LIN {X 0,Y 439.372,Z 569.757,A -85,B 0,C 180,E1 -9212.03,E2 -9212.03} C_VEL
LIN {X 0,Y 439.398,Z 569.751,A -85,B 0,C 180,E1 -9215.34,E2 -9215.34} C_VEL
LIN {X 0,Y 439.39,Z 569.756,A -85,B 0,C 180,E1 -9218.594,E2 -9218.594} C_VEL
LIN {X 0,Y 439.391,Z 569.751,A -85,B 0,C 180,E1 -9221.256,E2 -9221.256} C_VEL
LIN {X 0,Y 439.407,Z 569.752,A -85,B 0,C 180,E1 -9224.728,E2 -9224.728} C_VEL
LIN {X 0,Y 439.399,Z 569.751,A -85,B 0,C 180,E1 -9227.795,E2 -9227.795} C_VEL
LIN {X 0,Y 439.438,Z 569.749,A -85,B 0,C 180,E1 -9230.228,E2 -9230.228} C_VEL
LIN {X 0,Y 439.374,Z 569.754,A -85,B 0,C 180,E1 -9233.712,E2 -9233.712} C_VEL
LIN {X 0,Y 439.373,Z 569.756,A -85,B 0,C 180,E1 -9237.053,E2 -9237.053} C_VEL
LIN {X 0,Y 439.383,Z 569.755,A -85,B 0,C 180,E1 -9240.274,E2 -9240.274} C_VEL
LIN {X 0,Y 439.429,Z 569.747,A -85,B 0,C 180,E1 -9243.396,E2 -9243.396} C_VEL
LIN {X 0,Y 439.387,Z 569.755,A -85,B 0,C 180,E1 -9246.429,E2 -9246.429} C_VEL
LIN {X 0,Y 439.388,Z 569.751,A -85,B 0,C 180,E1 -9249.396,E2 -9249.396} C_VEL
LIN {X 0,Y 439.431,Z 569.749,A -85,B 0,C 180,E1 -9252.309,E2 -9252.309} C_VEL
LIN {X 0,Y 439.447,Z 569.746,A -85,B 0,C 180,E1 -9255.173,E2 -9255.173} C_VEL
LIN {X 0,Y 439.507,Z 569.738,A -85,B 0,C 180,E1 -9258.001,E2 -9258.001} C_VEL
LIN {X 0,Y 439.547,Z 569.733,A -85,B 0,C 180,E1 -9261.725,E2 -9261.725} C_VEL
LIN {X 0,Y 439.621,Z 569.726,A -85,B 0,C 180,E1 -9264.495,E2 -9264.495} C_VEL
LIN {X 0,Y 439.635,Z 569.724,A -85,B 0,C 180,E1 -9268.167,E2 -9268.167} C_VEL
LIN {X 0,Y 439.63,Z 569.725,A -85,B 0,C 180,E1 -9268.568,E2 -9268.568} C_VEL
LIN {X 0,Y 442.794,Z 580.936,A -85,B 0,C 180,E1 -9269.301,E2 -9269.301} C_VEL
LIN {X 0,Y 442.766,Z 587.106,A -85,B 0,C 180,E1 -9269.714,E2 -9269.714} C_VEL
LIN {X 0,Y 442.691,Z 589.675,A -85,B 0,C 180,E1 -9269.904,E2 -9269.904} C_VEL
LIN {X 0,Y 441.903,Z 594.784,A -85,B 0,C 180,E1 -9270.276,E2 -9270.276} C_VEL
LIN {X 0,Y 438.786,Z 602.936,A -85,B 0,C 180,E1 -9270.891,E2 -9270.891} C_VEL
LIN {X 0,Y 435.571,Z 610.599,A -85,B 0,C 180,E1 -9271.598,E2 -9271.598} C_VEL
LIN {X 0,Y 434.642,Z 614.939,A -85,B 0,C 180,E1 -9272.11,E2 -9272.11} C_VEL
LIN {X 0,Y 433.977,Z 624.554,A -85,B 0,C 180,E1 -9273.481,E2 -9273.481} C_VEL
LIN {X 0,Y 433.566,Z 632.408,A -85,B 0,C 180,E1 -9274.881,E2 -9274.881} C_VEL
LIN {X 0,Y 433.204,Z 637.758,A -85,B 0,C 180,E1 -9276.052,E2 -9276.052} C_VEL
LIN {X 0,Y 432.906,Z 642.988,A -85,B 0,C 180,E1 -9277.461,E2 -9277.461} C_VEL
LIN {X 0,Y 432.602,Z 647.086,A -85,B 0,C 180,E1 -9278.877,E2 -9278.877} C_VEL
LIN {X 0,Y 432.379,Z 650.136,A -85,B 0,C 180,E1 -9280.299,E2 -9280.299} C_VEL
LIN {X 0,Y 432.284,Z 651.639,A -85,B 0,C 180,E1 -9281.249,E2 -9281.249} C_VEL
LIN {X 0,Y 432.251,Z 653.107,A -85,B 0,C 180,E1 -9282.7,E2 -9282.7} C_VEL
LIN {X 0,Y 432.204,Z 653.639,A -85,B 0,C 180,E1 -9284.117,E2 -9284.117} C_VEL
LIN {X 0,Y 432.223,Z 653.484,A -85,B 0,C 180,E1 -9285.079,E2 -9285.079} C_VEL
LIN {X 0,Y 432.331,Z 652.582,A -85,B 0,C 180,E1 -9286.443,E2 -9286.443} C_VEL
LIN {X 0,Y 432.509,Z 650.537,A -85,B 0,C 180,E1 -9287.982,E2 -9287.982} C_VEL
LIN {X 0,Y 432.853,Z 646.995,A -85,B 0,C 180,E1 -9289.66,E2 -9289.66} C_VEL
LIN {X 0,Y 433.263,Z 641.799,A -85,B 0,C 180,E1 -9291.405,E2 -9291.405} C_VEL
LIN {X 0,Y 433.769,Z 635.934,A -85,B 0,C 180,E1 -9292.882,E2 -9292.882} C_VEL
LIN {X 0,Y 434.305,Z 628.458,A -85,B 0,C 180,E1 -9294.37,E2 -9294.37} C_VEL
LIN {X 0,Y 434.941,Z 620.541,A -85,B 0,C 180,E1 -9295.636,E2 -9295.636} C_VEL
LIN {X 0,Y 435.577,Z 611.178,A -85,B 0,C 180,E1 -9296.857,E2 -9296.857} C_VEL
LIN {X 0,Y 436.16,Z 600.306,A -85,B 0,C 180,E1 -9297.988,E2 -9297.988} C_VEL
LIN {X 0,Y 436.788,Z 589.714,A -85,B 0,C 180,E1 -9298.861,E2 -9298.861} C_VEL
LIN {X 0,Y 436.842,Z 584.716,A -85,B 0,C 180,E1 -9299.218,E2 -9299.218} C_VEL
LIN {X 0,Y 433.122,Z 573.093,A -85,B 0,C 180,E1 -9300.097,E2 -9300.097} C_VEL
LIN {X 0,Y 432.389,Z 570.629,A -85,B 0,C 180,E1 -9300.255,E2 -9300.255} C_VEL
LIN {X 0,Y 432.353,Z 570.628,A -85,B 0,C 180,E1 -9304.003,E2 -9304.003} C_VEL
LIN {X 0,Y 432.328,Z 570.635,A -85,B 0,C 180,E1 -9307.198,E2 -9307.198} C_VEL
LIN {X 0,Y 432.436,Z 570.815,A -85,B 0,C 180,E1 -9308.895,E2 -9308.895} C_VEL
LIN {X 0,Y 433.241,Z 576.214,A -85,B 0,C 180,E1 -9311.069,E2 -9311.069} C_VEL
LIN {X 0,Y 433.258,Z 582.668,A -85,B 0,C 180,E1 -9313.627,E2 -9313.627} C_VEL
LIN {X 0,Y 433.14,Z 590.995,A -85,B 0,C 180,E1 -9316.898,E2 -9316.898} C_VEL
LIN {X 0,Y 432.831,Z 599.434,A -85,B 0,C 180,E1 -9320.219,E2 -9320.219} C_VEL
LIN {X 0,Y 432.697,Z 606.671,A -85,B 0,C 180,E1 -9323.061,E2 -9323.061} C_VEL
LIN {X 0,Y 432.492,Z 615.337,A -85,B 0,C 180,E1 -9326.462,E2 -9326.462} C_VEL
LIN {X 0,Y 432.248,Z 623.677,A -85,B 0,C 180,E1 -9329.733,E2 -9329.733} C_VEL
LIN {X 0,Y 432.206,Z 625.589,A -85,B 0,C 180,E1 -9330.479,E2 -9330.479} C_VEL
LIN {X 0,Y 435.447,Z 641.385,A -85,B 0,C 180,E1 -9331.111,E2 -9331.111} C_VEL
LIN {X 0,Y 435.762,Z 646.126,A -85,B 0,C 180,E1 -9331.329,E2 -9331.329} C_VEL
LIN {X 0,Y 435.232,Z 658.171,A -85,B 0,C 180,E1 -9331.96,E2 -9331.96} C_VEL
LIN {X 0,Y 434.708,Z 669.886,A -85,B 0,C 180,E1 -9332.769,E2 -9332.769} C_VEL
LIN {X 0,Y 434.076,Z 680.526,A -85,B 0,C 180,E1 -9333.691,E2 -9333.691} C_VEL
LIN {X 0,Y 433.476,Z 690.924,A -85,B 0,C 180,E1 -9334.812,E2 -9334.812} C_VEL
LIN {X 0,Y 432.897,Z 700.253,A -85,B 0,C 180,E1 -9336.055,E2 -9336.055} C_VEL
LIN {X 0,Y 432.385,Z 708.024,A -85,B 0,C 180,E1 -9337.318,E2 -9337.318} C_VEL
LIN {X 0,Y 432.035,Z 715.276,A -85,B 0,C 180,E1 -9338.781,E2 -9338.781} C_VEL
LIN {X 0,Y 431.673,Z 721.759,A -85,B 0,C 180,E1 -9340.461,E2 -9340.461} C_VEL
LIN {X 0,Y 431.436,Z 726.172,A -85,B 0,C 180,E1 -9341.971,E2 -9341.971} C_VEL
LIN {X 0,Y 431.358,Z 728.335,A -85,B 0,C 180,E1 -9342.947,E2 -9342.947} C_VEL
LIN {X 0,Y 431.26,Z 730.235,A -85,B 0,C 180,E1 -9344.043,E2 -9344.043} C_VEL
LIN {X 0,Y 431.221,Z 731.301,A -85,B 0,C 180,E1 -9344.885,E2 -9344.885} C_VEL
LIN {X 0,Y 431.171,Z 732.08,A -85,B 0,C 180,E1 -9345.848,E2 -9345.848} C_VEL
LIN {X 0,Y 431.179,Z 732.449,A -85,B 0,C 180,E1 -9346.81,E2 -9346.81} C_VEL
LIN {X 0,Y 431.29,Z 732.372,A -85,B 0,C 180,E1 -9347.876,E2 -9347.876} C_VEL
LIN {X 0,Y 431.271,Z 731.013,A -85,B 0,C 180,E1 -9349.674,E2 -9349.674} C_VEL
LIN {X 0,Y 431.343,Z 729.708,A -85,B 0,C 180,E1 -9350.623,E2 -9350.623} C_VEL
LIN {X 0,Y 431.546,Z 726.899,A -85,B 0,C 180,E1 -9352.044,E2 -9352.044} C_VEL
LIN {X 0,Y 431.711,Z 723.065,A -85,B 0,C 180,E1 -9353.457,E2 -9353.457} C_VEL
LIN {X 0,Y 431.952,Z 718.085,A -85,B 0,C 180,E1 -9354.866,E2 -9354.866} C_VEL
LIN {X 0,Y 432.307,Z 711.79,A -85,B 0,C 180,E1 -9356.272,E2 -9356.272} C_VEL
LIN {X 0,Y 432.829,Z 703.98,A -85,B 0,C 180,E1 -9357.674,E2 -9357.674} C_VEL
LIN {X 0,Y 433.386,Z 696.051,A -85,B 0,C 180,E1 -9358.839,E2 -9358.839} C_VEL
LIN {X 0,Y 434.041,Z 686.397,A -85,B 0,C 180,E1 -9360,E2 -9360} C_VEL
LIN {X 0,Y 434.7,Z 675.647,A -85,B 0,C 180,E1 -9361.043,E2 -9361.043} C_VEL
LIN {X 0,Y 435.374,Z 663.66,A -85,B 0,C 180,E1 -9361.966,E2 -9361.966} C_VEL
LIN {X 0,Y 436.015,Z 650.788,A -85,B 0,C 180,E1 -9362.714,E2 -9362.714} C_VEL
LIN {X 0,Y 436.08,Z 643.477,A -85,B 0,C 180,E1 -9363.061,E2 -9363.061} C_VEL
LIN {X 0,Y 433.461,Z 631.54,A -85,B 0,C 180,E1 -9363.603,E2 -9363.603} C_VEL
LIN {X 0,Y 432.321,Z 627.329,A -85,B 0,C 180,E1 -9363.787,E2 -9363.787} C_VEL
LIN {X 0,Y 432.607,Z 622.657,A -85,B 0,C 180,E1 -9365.594,E2 -9365.594} C_VEL
LIN {X 0,Y 432.829,Z 614.137,A -85,B 0,C 180,E1 -9368.874,E2 -9368.874} C_VEL
LIN {X 0,Y 433.025,Z 606.775,A -85,B 0,C 180,E1 -9371.705,E2 -9371.705} C_VEL
LIN {X 0,Y 433.189,Z 599.173,A -85,B 0,C 180,E1 -9374.565,E2 -9374.565} C_VEL
LIN {X 0,Y 433.297,Z 591.196,A -85,B 0,C 180,E1 -9377.462,E2 -9377.462} C_VEL
LIN {X 0,Y 433.431,Z 582.92,A -85,B 0,C 180,E1 -9380.403,E2 -9380.403} C_VEL
LIN {X 0,Y 433.298,Z 575.774,A -85,B 0,C 180,E1 -9382.91,E2 -9382.91} C_VEL
LIN {X 0,Y 432.358,Z 570.636,A -85,B 0,C 180,E1 -9384.762,E2 -9384.762} C_VEL
LIN {X 0,Y 432.387,Z 570.629,A -85,B 0,C 180,E1 -9387.072,E2 -9387.072} C_VEL
LIN {X 0,Y 432.362,Z 570.631,A -85,B 0,C 180,E1 -9390.516,E2 -9390.516} C_VEL
LIN {X 0,Y 432.354,Z 570.631,A -85,B 0,C 180,E1 -9394.005,E2 -9394.005} C_VEL
LIN {X 0,Y 432.329,Z 570.633,A -85,B 0,C 180,E1 -9397.2,E2 -9397.2} C_VEL
LIN {X 0,Y 432.353,Z 570.629,A -85,B 0,C 180,E1 -9400.184,E2 -9400.184} C_VEL
LIN {X 0,Y 432.361,Z 570.63,A -85,B 0,C 180,E1 -9403.056,E2 -9403.056} C_VEL
LIN {X 0,Y 432.374,Z 570.63,A -85,B 0,C 180,E1 -9405.66,E2 -9405.66} C_VEL
LIN {X 0,Y 432.377,Z 570.803,A -85,B 0,C 180,E1 -9407.351,E2 -9407.351} C_VEL
LIN {X 0,Y 434.187,Z 579.301,A -85,B 0,C 180,E1 -9410.257,E2 -9410.257} C_VEL
LIN {X 0,Y 435.681,Z 587.385,A -85,B 0,C 180,E1 -9412.837,E2 -9412.837} C_VEL
LIN {X 0,Y 435.534,Z 593.083,A -85,B 0,C 180,E1 -9414.486,E2 -9414.486} C_VEL
LIN {X 0,Y 434.642,Z 604.82,A -85,B 0,C 180,E1 -9417.752,E2 -9417.752} C_VEL
LIN {X 0,Y 433.929,Z 616.968,A -85,B 0,C 180,E1 -9420.998,E2 -9420.998} C_VEL
LIN {X 0,Y 433.289,Z 629.663,A -85,B 0,C 180,E1 -9424.287,E2 -9424.287} C_VEL
LIN {X 0,Y 432.691,Z 643.56,A -85,B 0,C 180,E1 -9427.794,E2 -9427.794} C_VEL
LIN {X 0,Y 432.277,Z 657.625,A -85,B 0,C 180,E1 -9431.272,E2 -9431.272} C_VEL
LIN {X 0,Y 432.086,Z 665.28,A -85,B 0,C 180,E1 -9433.15,E2 -9433.15} C_VEL
LIN {X 0,Y 433.733,Z 681.12,A -85,B 0,C 180,E1 -9433.658,E2 -9433.658} C_VEL
LIN {X 0,Y 434.619,Z 693.584,A -85,B 0,C 180,E1 -9434.226,E2 -9434.226} C_VEL
LIN {X 0,Y 435.052,Z 699.186,A -85,B 0,C 180,E1 -9434.542,E2 -9434.542} C_VEL
LIN {X 0,Y 434.161,Z 715.758,A -85,B 0,C 180,E1 -9435.59,E2 -9435.59} C_VEL
LIN {X 0,Y 433.491,Z 727,A -85,B 0,C 180,E1 -9436.507,E2 -9436.507} C_VEL
LIN {X 0,Y 432.961,Z 737.61,A -85,B 0,C 180,E1 -9437.581,E2 -9437.581} C_VEL
LIN {X 0,Y 432.469,Z 747.017,A -85,B 0,C 180,E1 -9438.756,E2 -9438.756} C_VEL
LIN {X 0,Y 431.986,Z 756.151,A -85,B 0,C 180,E1 -9440.165,E2 -9440.165} C_VEL
LIN {X 0,Y 431.714,Z 763.519,A -85,B 0,C 180,E1 -9441.576,E2 -9441.576} C_VEL
LIN {X 0,Y 431.516,Z 769.377,A -85,B 0,C 180,E1 -9442.985,E2 -9442.985} C_VEL
LIN {X 0,Y 431.451,Z 773.978,A -85,B 0,C 180,E1 -9444.392,E2 -9444.392} C_VEL
LIN {X 0,Y 431.397,Z 776.404,A -85,B 0,C 180,E1 -9445.329,E2 -9445.329} C_VEL
LIN {X 0,Y 431.377,Z 778.39,A -85,B 0,C 180,E1 -9446.264,E2 -9446.264} C_VEL
LIN {X 0,Y 431.407,Z 779.895,A -85,B 0,C 180,E1 -9447.2,E2 -9447.2} C_VEL
LIN {X 0,Y 431.405,Z 780.964,A -85,B 0,C 180,E1 -9448.134,E2 -9448.134} C_VEL
LIN {X 0,Y 431.402,Z 781.628,A -85,B 0,C 180,E1 -9449.067,E2 -9449.067} C_VEL
LIN {X 0,Y 431.382,Z 781.873,A -85,B 0,C 180,E1 -9450.001,E2 -9450.001} C_VEL
LIN {X 0,Y 431.401,Z 781.664,A -85,B 0,C 180,E1 -9450.934,E2 -9450.934} C_VEL
LIN {X 0,Y 431.407,Z 781.049,A -85,B 0,C 180,E1 -9451.868,E2 -9451.868} C_VEL
LIN {X 0,Y 431.406,Z 780.029,A -85,B 0,C 180,E1 -9452.802,E2 -9452.802} C_VEL
LIN {X 0,Y 431.36,Z 778.542,A -85,B 0,C 180,E1 -9453.737,E2 -9453.737} C_VEL
LIN {X 0,Y 431.445,Z 775.484,A -85,B 0,C 180,E1 -9455.141,E2 -9455.141} C_VEL
LIN {X 0,Y 431.445,Z 771.315,A -85,B 0,C 180,E1 -9456.548,E2 -9456.548} C_VEL
LIN {X 0,Y 431.65,Z 764.913,A -85,B 0,C 180,E1 -9458.191,E2 -9458.191} C_VEL
LIN {X 0,Y 431.93,Z 757.897,A -85,B 0,C 180,E1 -9459.601,E2 -9459.601} C_VEL
LIN {X 0,Y 432.355,Z 749.061,A -85,B 0,C 180,E1 -9461.012,E2 -9461.012} C_VEL
LIN {X 0,Y 432.872,Z 739.007,A -85,B 0,C 180,E1 -9462.305,E2 -9462.305} C_VEL
LIN {X 0,Y 433.409,Z 728.753,A -85,B 0,C 180,E1 -9463.359,E2 -9463.359} C_VEL
LIN {X 0,Y 434.093,Z 717.383,A -85,B 0,C 180,E1 -9464.295,E2 -9464.295} C_VEL
LIN {X 0,Y 434.676,Z 705.557,A -85,B 0,C 180,E1 -9465.053,E2 -9465.053} C_VEL
LIN {X 0,Y 434.802,Z 696.334,A -85,B 0,C 180,E1 -9465.529,E2 -9465.529} C_VEL
LIN {X 0,Y 433.813,Z 685.114,A -85,B 0,C 180,E1 -9466.063,E2 -9466.063} C_VEL
LIN {X 0,Y 432.601,Z 671.595,A -85,B 0,C 180,E1 -9466.526,E2 -9466.526} C_VEL
LIN {X 0,Y 432.071,Z 666.093,A -85,B 0,C 180,E1 -9466.682,E2 -9466.682} C_VEL
LIN {X 0,Y 432.394,Z 652.62,A -85,B 0,C 180,E1 -9469.958,E2 -9469.958} C_VEL
LIN {X 0,Y 432.844,Z 638.506,A -85,B 0,C 180,E1 -9473.442,E2 -9473.442} C_VEL
LIN {X 0,Y 433.472,Z 624.3,A -85,B 0,C 180,E1 -9476.999,E2 -9476.999} C_VEL
LIN {X 0,Y 434.144,Z 610.513,A -85,B 0,C 180,E1 -9480.521,E2 -9480.521} C_VEL
LIN {X 0,Y 434.876,Z 596.628,A -85,B 0,C 180,E1 -9484.167,E2 -9484.167} C_VEL
LIN {X 0,Y 435.346,Z 587.383,A -85,B 0,C 180,E1 -9486.678,E2 -9486.678} C_VEL
LIN {X 0,Y 434.429,Z 581.267,A -85,B 0,C 180,E1 -9488.446,E2 -9488.446} C_VEL
LIN {X 0,Y 432.378,Z 570.63,A -85,B 0,C 180,E1 -9491.727,E2 -9491.727} C_VEL
LIN {X 0,Y 432.339,Z 570.634,A -85,B 0,C 180,E1 -9494.347,E2 -9494.347} C_VEL
LIN {X 0,Y 432.325,Z 570.635,A -85,B 0,C 180,E1 -9497.016,E2 -9497.016} C_VEL
LIN {X 0,Y 432.346,Z 570.631,A -85,B 0,C 180,E1 -9499.82,E2 -9499.82} C_VEL
LIN {X 0,Y 432.32,Z 570.632,A -85,B 0,C 180,E1 -9503.023,E2 -9503.023} C_VEL
LIN {X 0,Y 432.365,Z 570.629,A -85,B 0,C 180,E1 -9505.996,E2 -9505.996} C_VEL
LIN {X 0,Y 432.352,Z 570.629,A -85,B 0,C 180,E1 -9509.49,E2 -9509.49} C_VEL
LIN {X 0,Y 432.396,Z 570.624,A -85,B 0,C 180,E1 -9512.928,E2 -9512.928} C_VEL
LIN {X 0,Y 432.376,Z 570.628,A -85,B 0,C 180,E1 -9516.023,E2 -9516.023} C_VEL
LIN {X 0,Y 432.355,Z 570.629,A -85,B 0,C 180,E1 -9519.046,E2 -9519.046} C_VEL
LIN {X 0,Y 432.383,Z 570.627,A -85,B 0,C 180,E1 -9522.011,E2 -9522.011} C_VEL
LIN {X 0,Y 432.4,Z 570.623,A -85,B 0,C 180,E1 -9524.926,E2 -9524.926} C_VEL
LIN {X 0,Y 432.463,Z 570.616,A -85,B 0,C 180,E1 -9527.803,E2 -9527.803} C_VEL
LIN {X 0,Y 432.496,Z 570.61,A -85,B 0,C 180,E1 -9531.59,E2 -9531.59} C_VEL
LIN {X 0,Y 432.601,Z 570.601,A -85,B 0,C 180,E1 -9534.406,E2 -9534.406} C_VEL
LIN {X 0,Y 432.607,Z 570.6,A -85,B 0,C 180,E1 -9538.138,E2 -9538.138} C_VEL
LIN {X 0,Y 432.737,Z 570.582,A -85,B 0,C 180,E1 -9540,E2 -9540} C_VEL
LIN {X 0,Y 432.595,Z 570.6,A -85,B 0,C 180,E1 -9542.793,E2 -9542.793} C_VEL
LIN {X 0,Y 432.576,Z 570.604,A -85,B 0,C 180,E1 -9546.53,E2 -9546.53} C_VEL
LIN {X 0,Y 432.446,Z 570.617,A -85,B 0,C 180,E1 -9549.353,E2 -9549.353} C_VEL
LIN {X 0,Y 432.434,Z 570.62,A -85,B 0,C 180,E1 -9552.803,E2 -9552.803} C_VEL
LIN {X 0,Y 432.416,Z 570.624,A -85,B 0,C 180,E1 -9556.478,E2 -9556.478} C_VEL
LIN {X 0,Y 432.342,Z 570.632,A -85,B 0,C 180,E1 -9559.96,E2 -9559.96} C_VEL
LIN {X 0,Y 432.322,Z 570.634,A -85,B 0,C 180,E1 -9562.964,E2 -9562.964} C_VEL
LIN {X 0,Y 432.367,Z 570.629,A -85,B 0,C 180,E1 -9566.032,E2 -9566.032} C_VEL
LIN {X 0,Y 432.345,Z 570.63,A -85,B 0,C 180,E1 -9569.187,E2 -9569.187} C_VEL
LIN {X 0,Y 432.325,Z 570.635,A -85,B 0,C 180,E1 -9572.442,E2 -9572.442} C_VEL
LIN {X 0,Y 432.347,Z 570.629,A -85,B 0,C 180,E1 -9575.632,E2 -9575.632} C_VEL
LIN {X 0,Y 432.352,Z 570.631,A -85,B 0,C 180,E1 -9578.716,E2 -9578.716} C_VEL
LIN {X 0,Y 432.336,Z 570.63,A -85,B 0,C 180,E1 -9581.796,E2 -9581.796} C_VEL
LIN {X 0,Y 432.342,Z 570.633,A -85,B 0,C 180,E1 -9584.346,E2 -9584.346} C_VEL
LIN {X 0,Y 432.326,Z 570.633,A -85,B 0,C 180,E1 -9587.014,E2 -9587.014} C_VEL
LIN {X 0,Y 432.342,Z 570.63,A -85,B 0,C 180,E1 -9589.819,E2 -9589.819} C_VEL
LIN {X 0,Y 432.307,Z 570.636,A -85,B 0,C 180,E1 -9593.021,E2 -9593.021} C_VEL
LIN {X 0,Y 432.36,Z 570.628,A -85,B 0,C 180,E1 -9595.996,E2 -9595.996} C_VEL
LIN {X 0,Y 432.348,Z 570.629,A -85,B 0,C 180,E1 -9599.489,E2 -9599.489} C_VEL
LIN {X 0,Y 432.391,Z 570.626,A -85,B 0,C 180,E1 -9602.928,E2 -9602.928} C_VEL
LIN {X 0,Y 432.372,Z 570.628,A -85,B 0,C 180,E1 -9606.023,E2 -9606.023} C_VEL
LIN {X 0,Y 432.35,Z 570.63,A -85,B 0,C 180,E1 -9609.045,E2 -9609.045} C_VEL
LIN {X 0,Y 432.378,Z 570.626,A -85,B 0,C 180,E1 -9612.01,E2 -9612.01} C_VEL
LIN {X 0,Y 432.395,Z 570.625,A -85,B 0,C 180,E1 -9614.926,E2 -9614.926} C_VEL
LIN {X 0,Y 432.48,Z 570.612,A -85,B 0,C 180,E1 -9617.803,E2 -9617.803} C_VEL
LIN {X 0,Y 432.491,Z 570.611,A -85,B 0,C 180,E1 -9621.59,E2 -9621.59} C_VEL
LIN {X 0,Y 432.597,Z 570.602,A -85,B 0,C 180,E1 -9624.405,E2 -9624.405} C_VEL
LIN {X 0,Y 432.608,Z 570.599,A -85,B 0,C 180,E1 -9628.254,E2 -9628.254} C_VEL
LIN {X 0,Y 432.606,Z 570.599,A -85,B 0,C 180,E1 -9628.341,E2 -9628.341} C_VEL
LIN {X 0,Y 436.064,Z 582.901,A -85,B 0,C 180,E1 -9629.165,E2 -9629.165} C_VEL
LIN {X 0,Y 435.704,Z 594.325,A -85,B 0,C 180,E1 -9629.999,E2 -9629.999} C_VEL
LIN {X 0,Y 435.133,Z 605.628,A -85,B 0,C 180,E1 -9631.04,E2 -9631.04} C_VEL
LIN {X 0,Y 434.642,Z 614.939,A -85,B 0,C 180,E1 -9632.11,E2 -9632.11} C_VEL
LIN {X 0,Y 433.727,Z 619.196,A -85,B 0,C 180,E1 -9632.65,E2 -9632.65} C_VEL
LIN {X 0,Y 430.524,Z 625.776,A -85,B 0,C 180,E1 -9633.532,E2 -9633.532} C_VEL
LIN {X 0,Y 427.355,Z 631.843,A -85,B 0,C 180,E1 -9634.485,E2 -9634.485} C_VEL
LIN {X 0,Y 426.498,Z 635.132,A -85,B 0,C 180,E1 -9635.13,E2 -9635.13} C_VEL
LIN {X 0,Y 426.067,Z 641.369,A -85,B 0,C 180,E1 -9636.63,E2 -9636.63} C_VEL
LIN {X 0,Y 425.762,Z 645.694,A -85,B 0,C 180,E1 -9637.943,E2 -9637.943} C_VEL
LIN {X 0,Y 425.47,Z 649.65,A -85,B 0,C 180,E1 -9639.507,E2 -9639.507} C_VEL
LIN {X 0,Y 425.33,Z 651.503,A -85,B 0,C 180,E1 -9640.471,E2 -9640.471} C_VEL
LIN {X 0,Y 425.259,Z 653.863,A -85,B 0,C 180,E1 -9642.405,E2 -9642.405} C_VEL
LIN {X 0,Y 425.196,Z 654.474,A -85,B 0,C 180,E1 -9643.379,E2 -9643.379} C_VEL
LIN {X 0,Y 425.196,Z 654.647,A -85,B 0,C 180,E1 -9644.354,E2 -9644.354} C_VEL
LIN {X 0,Y 425.21,Z 654.407,A -85,B 0,C 180,E1 -9645.333,E2 -9645.333} C_VEL
LIN {X 0,Y 425.331,Z 653.521,A -85,B 0,C 180,E1 -9646.592,E2 -9646.592} C_VEL
LIN {X 0,Y 425.555,Z 651.19,A -85,B 0,C 180,E1 -9648.286,E2 -9648.286} C_VEL
LIN {X 0,Y 425.9,Z 647.859,A -85,B 0,C 180,E1 -9649.851,E2 -9649.851} C_VEL
LIN {X 0,Y 426.23,Z 643.782,A -85,B 0,C 180,E1 -9651.268,E2 -9651.268} C_VEL
LIN {X 0,Y 426.83,Z 637.536,A -85,B 0,C 180,E1 -9652.931,E2 -9652.931} C_VEL
LIN {X 0,Y 427.443,Z 629.728,A -85,B 0,C 180,E1 -9654.528,E2 -9654.528} C_VEL
LIN {X 0,Y 428.048,Z 622.381,A -85,B 0,C 180,E1 -9655.738,E2 -9655.738} C_VEL
LIN {X 0,Y 428.769,Z 612.584,A -85,B 0,C 180,E1 -9657.054,E2 -9657.054} C_VEL
LIN {X 0,Y 429.375,Z 602.358,A -85,B 0,C 180,E1 -9658.15,E2 -9658.15} C_VEL
LIN {X 0,Y 430.053,Z 591.346,A -85,B 0,C 180,E1 -9659.089,E2 -9659.089} C_VEL
LIN {X 0,Y 430.227,Z 587.846,A -85,B 0,C 180,E1 -9659.344,E2 -9659.344} C_VEL
LIN {X 0,Y 429.021,Z 582.892,A -85,B 0,C 180,E1 -9659.749,E2 -9659.749} C_VEL
LIN {X 0,Y 425.323,Z 571.505,A -85,B 0,C 180,E1 -9660.608,E2 -9660.608} C_VEL
LIN {X 0,Y 425.305,Z 571.507,A -85,B 0,C 180,E1 -9664.287,E2 -9664.287} C_VEL
LIN {X 0,Y 425.289,Z 571.511,A -85,B 0,C 180,E1 -9667.692,E2 -9667.692} C_VEL
LIN {X 0,Y 425.344,Z 571.596,A -85,B 0,C 180,E1 -9668.665,E2 -9668.665} C_VEL
LIN {X 0,Y 426.115,Z 576.426,A -85,B 0,C 180,E1 -9670.652,E2 -9670.652} C_VEL
LIN {X 0,Y 426.318,Z 581.161,A -85,B 0,C 180,E1 -9672.522,E2 -9672.522} C_VEL
LIN {X 0,Y 426.183,Z 589.045,A -85,B 0,C 180,E1 -9675.662,E2 -9675.662} C_VEL
LIN {X 0,Y 425.943,Z 596.747,A -85,B 0,C 180,E1 -9678.701,E2 -9678.701} C_VEL
LIN {X 0,Y 425.727,Z 606.096,A -85,B 0,C 180,E1 -9682.408,E2 -9682.408} C_VEL
LIN {X 0,Y 425.527,Z 614.769,A -85,B 0,C 180,E1 -9685.838,E2 -9685.838} C_VEL
LIN {X 0,Y 425.273,Z 623.41,A -85,B 0,C 180,E1 -9689.241,E2 -9689.241} C_VEL
LIN {X 0,Y 425.212,Z 626.135,A -85,B 0,C 180,E1 -9690.245,E2 -9690.245} C_VEL
LIN {X 0,Y 428.03,Z 639.809,A -85,B 0,C 180,E1 -9690.782,E2 -9690.782} C_VEL
LIN {X 0,Y 428.914,Z 645.393,A -85,B 0,C 180,E1 -9691.052,E2 -9691.052} C_VEL
LIN {X 0,Y 428.366,Z 658.428,A -85,B 0,C 180,E1 -9691.737,E2 -9691.737} C_VEL
LIN {X 0,Y 427.758,Z 670.823,A -85,B 0,C 180,E1 -9692.611,E2 -9692.611} C_VEL
LIN {X 0,Y 427.04,Z 682.091,A -85,B 0,C 180,E1 -9693.619,E2 -9693.619} C_VEL
LIN {X 0,Y 426.428,Z 692.398,A -85,B 0,C 180,E1 -9694.779,E2 -9694.779} C_VEL
LIN {X 0,Y 425.803,Z 702.257,A -85,B 0,C 180,E1 -9696.148,E2 -9696.148} C_VEL
LIN {X 0,Y 425.245,Z 710.875,A -85,B 0,C 180,E1 -9697.659,E2 -9697.659} C_VEL
LIN {X 0,Y 424.871,Z 717.742,A -85,B 0,C 180,E1 -9699.168,E2 -9699.168} C_VEL
LIN {X 0,Y 424.567,Z 723.08,A -85,B 0,C 180,E1 -9700.667,E2 -9700.667} C_VEL
LIN {X 0,Y 424.349,Z 727.135,A -85,B 0,C 180,E1 -9702.158,E2 -9702.158} C_VEL
LIN {X 0,Y 424.202,Z 730.493,A -85,B 0,C 180,E1 -9703.924,E2 -9703.924} C_VEL
LIN {X 0,Y 424.088,Z 732.353,A -85,B 0,C 180,E1 -9705.607,E2 -9705.607} C_VEL
LIN {X 0,Y 424.093,Z 732.81,A -85,B 0,C 180,E1 -9706.585,E2 -9706.585} C_VEL
LIN {X 0,Y 424.19,Z 732.82,A -85,B 0,C 180,E1 -9707.821,E2 -9707.821} C_VEL
LIN {X 0,Y 424.203,Z 731.696,A -85,B 0,C 180,E1 -9709.5,E2 -9709.5} C_VEL
LIN {X 0,Y 424.257,Z 730.472,A -85,B 0,C 180,E1 -9710.465,E2 -9710.465} C_VEL
LIN {X 0,Y 424.447,Z 727.825,A -85,B 0,C 180,E1 -9711.91,E2 -9711.91} C_VEL
LIN {X 0,Y 424.657,Z 724.157,A -85,B 0,C 180,E1 -9713.348,E2 -9713.348} C_VEL
LIN {X 0,Y 424.885,Z 719.389,A -85,B 0,C 180,E1 -9714.781,E2 -9714.781} C_VEL
LIN {X 0,Y 425.257,Z 713.37,A -85,B 0,C 180,E1 -9716.21,E2 -9716.21} C_VEL
LIN {X 0,Y 425.801,Z 705.834,A -85,B 0,C 180,E1 -9717.635,E2 -9717.635} C_VEL
LIN {X 0,Y 426.477,Z 696.482,A -85,B 0,C 180,E1 -9719.056,E2 -9719.056} C_VEL
LIN {X 0,Y 427.188,Z 686.811,A -85,B 0,C 180,E1 -9720.236,E2 -9720.236} C_VEL
LIN {X 0,Y 427.888,Z 676.057,A -85,B 0,C 180,E1 -9721.294,E2 -9721.294} C_VEL
LIN {X 0,Y 428.576,Z 664.076,A -85,B 0,C 180,E1 -9722.232,E2 -9722.232} C_VEL
LIN {X 0,Y 429.181,Z 652.649,A -85,B 0,C 180,E1 -9722.919,E2 -9722.919} C_VEL
LIN {X 0,Y 429.403,Z 645.21,A -85,B 0,C 180,E1 -9723.284,E2 -9723.284} C_VEL
LIN {X 0,Y 426.766,Z 633.01,A -85,B 0,C 180,E1 -9723.881,E2 -9723.881} C_VEL
LIN {X 0,Y 425.455,Z 627.764,A -85,B 0,C 180,E1 -9724.115,E2 -9724.115} C_VEL
LIN {X 0,Y 425.668,Z 621.295,A -85,B 0,C 180,E1 -9726.637,E2 -9726.637} C_VEL
LIN {X 0,Y 425.915,Z 613.92,A -85,B 0,C 180,E1 -9729.498,E2 -9729.498} C_VEL
LIN {X 0,Y 426.171,Z 605.243,A -85,B 0,C 180,E1 -9732.864,E2 -9732.864} C_VEL
LIN {X 0,Y 426.332,Z 596.136,A -85,B 0,C 180,E1 -9736.275,E2 -9736.275} C_VEL
LIN {X 0,Y 426.448,Z 587.95,A -85,B 0,C 180,E1 -9739.245,E2 -9739.245} C_VEL
LIN {X 0,Y 426.569,Z 579.496,A -85,B 0,C 180,E1 -9742.268,E2 -9742.268} C_VEL
LIN {X 0,Y 426.095,Z 575.197,A -85,B 0,C 180,E1 -9743.835,E2 -9743.835} C_VEL
LIN {X 0,Y 425.303,Z 571.514,A -85,B 0,C 180,E1 -9745.228,E2 -9745.228} C_VEL
LIN {X 0,Y 425.344,Z 571.506,A -85,B 0,C 180,E1 -9747.558,E2 -9747.558} C_VEL
LIN {X 0,Y 425.291,Z 571.512,A -85,B 0,C 180,E1 -9750.816,E2 -9750.816} C_VEL
LIN {X 0,Y 425.306,Z 571.509,A -85,B 0,C 180,E1 -9754.289,E2 -9754.289} C_VEL
LIN {X 0,Y 425.283,Z 571.513,A -85,B 0,C 180,E1 -9757.694,E2 -9757.694} C_VEL
LIN {X 0,Y 425.298,Z 571.509,A -85,B 0,C 180,E1 -9760.525,E2 -9760.525} C_VEL
LIN {X 0,Y 425.328,Z 571.507,A -85,B 0,C 180,E1 -9763.363,E2 -9763.363} C_VEL
LIN {X 0,Y 425.335,Z 571.576,A -85,B 0,C 180,E1 -9766.9,E2 -9766.9} C_VEL
LIN {X 0,Y 427.248,Z 580.689,A -85,B 0,C 180,E1 -9770.096,E2 -9770.096} C_VEL
LIN {X 0,Y 428.704,Z 588.589,A -85,B 0,C 180,E1 -9772.66,E2 -9772.66} C_VEL
LIN {X 0,Y 428.728,Z 592.47,A -85,B 0,C 180,E1 -9773.835,E2 -9773.835} C_VEL
LIN {X 0,Y 427.867,Z 603.214,A -85,B 0,C 180,E1 -9776.9,E2 -9776.9} C_VEL
LIN {X 0,Y 427.046,Z 616.003,A -85,B 0,C 180,E1 -9780.416,E2 -9780.416} C_VEL
LIN {X 0,Y 426.355,Z 627.878,A -85,B 0,C 180,E1 -9783.574,E2 -9783.574} C_VEL
LIN {X 0,Y 425.796,Z 639.814,A -85,B 0,C 180,E1 -9786.664,E2 -9786.664} C_VEL
LIN {X 0,Y 425.311,Z 653.343,A -85,B 0,C 180,E1 -9790.104,E2 -9790.104} C_VEL
LIN {X 0,Y 425.052,Z 664.448,A -85,B 0,C 180,E1 -9792.852,E2 -9792.852} C_VEL
LIN {X 0,Y 426.577,Z 677.953,A -85,B 0,C 180,E1 -9793.275,E2 -9793.275} C_VEL
LIN {X 0,Y 427.411,Z 690.576,A -85,B 0,C 180,E1 -9793.83,E2 -9793.83} C_VEL
LIN {X 0,Y 428.117,Z 698.582,A -85,B 0,C 180,E1 -9794.285,E2 -9794.285} C_VEL
LIN {X 0,Y 427.431,Z 712.274,A -85,B 0,C 180,E1 -9795.114,E2 -9795.114} C_VEL
LIN {X 0,Y 426.737,Z 724.398,A -85,B 0,C 180,E1 -9796.064,E2 -9796.064} C_VEL
LIN {X 0,Y 426.136,Z 735.168,A -85,B 0,C 180,E1 -9797.136,E2 -9797.136} C_VEL
LIN {X 0,Y 425.553,Z 744.931,A -85,B 0,C 180,E1 -9798.329,E2 -9798.329} C_VEL
LIN {X 0,Y 425.037,Z 752.958,A -85,B 0,C 180,E1 -9799.521,E2 -9799.521} C_VEL
LIN {X 0,Y 424.728,Z 760.826,A -85,B 0,C 180,E1 -9800.957,E2 -9800.957} C_VEL
LIN {X 0,Y 424.473,Z 767.154,A -85,B 0,C 180,E1 -9802.389,E2 -9802.389} C_VEL
LIN {X 0,Y 424.319,Z 772.387,A -85,B 0,C 180,E1 -9803.891,E2 -9803.891} C_VEL
LIN {X 0,Y 424.326,Z 776.009,A -85,B 0,C 180,E1 -9805.251,E2 -9805.251} C_VEL
LIN {X 0,Y 424.28,Z 777.994,A -85,B 0,C 180,E1 -9806.202,E2 -9806.202} C_VEL
LIN {X 0,Y 424.334,Z 779.494,A -85,B 0,C 180,E1 -9807.153,E2 -9807.153} C_VEL
LIN {X 0,Y 424.32,Z 780.561,A -85,B 0,C 180,E1 -9808.103,E2 -9808.103} C_VEL
LIN {X 0,Y 424.339,Z 781.226,A -85,B 0,C 180,E1 -9809.052,E2 -9809.052} C_VEL
LIN {X 0,Y 424.318,Z 781.462,A -85,B 0,C 180,E1 -9810.001,E2 -9810.001} C_VEL
LIN {X 0,Y 424.338,Z 781.246,A -85,B 0,C 180,E1 -9810.95,E2 -9810.95} C_VEL
LIN {X 0,Y 424.322,Z 780.625,A -85,B 0,C 180,E1 -9811.899,E2 -9811.899} C_VEL
LIN {X 0,Y 424.331,Z 779.599,A -85,B 0,C 180,E1 -9812.849,E2 -9812.849} C_VEL
LIN {X 0,Y 424.265,Z 778.097,A -85,B 0,C 180,E1 -9813.8,E2 -9813.8} C_VEL
LIN {X 0,Y 424.374,Z 775.022,A -85,B 0,C 180,E1 -9815.227,E2 -9815.227} C_VEL
LIN {X 0,Y 424.359,Z 770.828,A -85,B 0,C 180,E1 -9816.658,E2 -9816.658} C_VEL
LIN {X 0,Y 424.601,Z 764.4,A -85,B 0,C 180,E1 -9818.328,E2 -9818.328} C_VEL
LIN {X 0,Y 424.894,Z 757.341,A -85,B 0,C 180,E1 -9819.762,E2 -9819.762} C_VEL
LIN {X 0,Y 425.344,Z 748.469,A -85,B 0,C 180,E1 -9821.196,E2 -9821.196} C_VEL
LIN {X 0,Y 425.82,Z 739.372,A -85,B 0,C 180,E1 -9822.391,E2 -9822.391} C_VEL
LIN {X 0,Y 426.407,Z 729.1,A -85,B 0,C 180,E1 -9823.483,E2 -9823.483} C_VEL
LIN {X 0,Y 427.085,Z 718.184,A -85,B 0,C 180,E1 -9824.413,E2 -9824.413} C_VEL
LIN {X 0,Y 427.622,Z 707.713,A -85,B 0,C 180,E1 -9825.125,E2 -9825.125} C_VEL
LIN {X 0,Y 427.945,Z 697.833,A -85,B 0,C 180,E1 -9825.662,E2 -9825.662} C_VEL
LIN {X 0,Y 426.731,Z 684.151,A -85,B 0,C 180,E1 -9826.307,E2 -9826.307} C_VEL
LIN {X 0,Y 425.577,Z 670.904,A -85,B 0,C 180,E1 -9826.771,E2 -9826.771} C_VEL
LIN {X 0,Y 424.981,Z 665.14,A -85,B 0,C 180,E1 -9826.924,E2 -9826.924} C_VEL
LIN {X 0,Y 425.307,Z 653.175,A -85,B 0,C 180,E1 -9829.9,E2 -9829.9} C_VEL
LIN {X 0,Y 425.762,Z 639.478,A -85,B 0,C 180,E1 -9833.339,E2 -9833.339} C_VEL
LIN {X 0,Y 426.368,Z 625.931,A -85,B 0,C 180,E1 -9836.783,E2 -9836.783} C_VEL
LIN {X 0,Y 427.119,Z 611.032,A -85,B 0,C 180,E1 -9840.67,E2 -9840.67} C_VEL
LIN {X 0,Y 427.817,Z 598.719,A -85,B 0,C 180,E1 -9843.955,E2 -9843.955} C_VEL
LIN {X 0,Y 428.361,Z 589.489,A -85,B 0,C 180,E1 -9846.492,E2 -9846.492} C_VEL
LIN {X 0,Y 427.832,Z 584.469,A -85,B 0,C 180,E1 -9847.954,E2 -9847.954} C_VEL
LIN {X 0,Y 425.719,Z 573.506,A -85,B 0,C 180,E1 -9851.327,E2 -9851.327} C_VEL
LIN {X 0,Y 425.311,Z 571.509,A -85,B 0,C 180,E1 -9852.021,E2 -9852.021} C_VEL
LIN {X 0,Y 425.29,Z 571.512,A -85,B 0,C 180,E1 -9855.283,E2 -9855.283} C_VEL
LIN {X 0,Y 425.28,Z 571.512,A -85,B 0,C 180,E1 -9858.622,E2 -9858.622} C_VEL
LIN {X 0,Y 425.32,Z 571.505,A -85,B 0,C 180,E1 -9861.103,E2 -9861.103} C_VEL
LIN {X 0,Y 425.306,Z 571.509,A -85,B 0,C 180,E1 -9864.664,E2 -9864.664} C_VEL
LIN {X 0,Y 425.27,Z 571.513,A -85,B 0,C 180,E1 -9868.073,E2 -9868.073} C_VEL
LIN {X 0,Y 425.336,Z 571.501,A -85,B 0,C 180,E1 -9871.368,E2 -9871.368} C_VEL
LIN {X 0,Y 425.3,Z 571.51,A -85,B 0,C 180,E1 -9874.555,E2 -9874.555} C_VEL
LIN {X 0,Y 425.292,Z 571.508,A -85,B 0,C 180,E1 -9877.661,E2 -9877.661} C_VEL
LIN {X 0,Y 425.367,Z 571.501,A -85,B 0,C 180,E1 -9880.704,E2 -9880.704} C_VEL
LIN {X 0,Y 425.393,Z 571.496,A -85,B 0,C 180,E1 -9883.688,E2 -9883.688} C_VEL
LIN {X 0,Y 425.416,Z 571.493,A -85,B 0,C 180,E1 -9887.598,E2 -9887.598} C_VEL
LIN {X 0,Y 425.447,Z 571.488,A -85,B 0,C 180,E1 -9891.45,E2 -9891.45} C_VEL
LIN {X 0,Y 425.558,Z 571.479,A -85,B 0,C 180,E1 -9894.313,E2 -9894.313} C_VEL
LIN {X 0,Y 425.576,Z 571.476,A -85,B 0,C 180,E1 -9898.107,E2 -9898.107} C_VEL
LIN {X 0,Y 425.707,Z 571.458,A -85,B 0,C 180,E1 -9900,E2 -9900} C_VEL
LIN {X 0,Y 425.548,Z 571.478,A -85,B 0,C 180,E1 -9902.84,E2 -9902.84} C_VEL
LIN {X 0,Y 425.535,Z 571.481,A -85,B 0,C 180,E1 -9906.638,E2 -9906.638} C_VEL
LIN {X 0,Y 425.404,Z 571.494,A -85,B 0,C 180,E1 -9909.509,E2 -9909.509} C_VEL
LIN {X 0,Y 425.397,Z 571.496,A -85,B 0,C 180,E1 -9912.903,E2 -9912.903} C_VEL
LIN {X 0,Y 425.365,Z 571.502,A -85,B 0,C 180,E1 -9916.605,E2 -9916.605} C_VEL
LIN {X 0,Y 425.331,Z 571.503,A -85,B 0,C 180,E1 -9919.635,E2 -9919.635} C_VEL
LIN {X 0,Y 425.31,Z 571.506,A -85,B 0,C 180,E1 -9923.365,E2 -9923.365} C_VEL
LIN {X 0,Y 425.349,Z 571.503,A -85,B 0,C 180,E1 -9926.844,E2 -9926.844} C_VEL
LIN {X 0,Y 425.293,Z 571.508,A -85,B 0,C 180,E1 -9929.719,E2 -9929.719} C_VEL
LIN {X 0,Y 425.284,Z 571.51,A -85,B 0,C 180,E1 -9933.047,E2 -9933.047} C_VEL
LIN {X 0,Y 425.287,Z 571.509,A -85,B 0,C 180,E1 -9935.929,E2 -9935.929} C_VEL
LIN {X 0,Y 425.3,Z 571.508,A -85,B 0,C 180,E1 -9939.043,E2 -9939.043} C_VEL
LIN {X 0,Y 425.279,Z 571.513,A -85,B 0,C 180,E1 -9942.652,E2 -9942.652} C_VEL
LIN {X 0,Y 425.27,Z 571.513,A -85,B 0,C 180,E1 -9946.044,E2 -9946.044} C_VEL
LIN {X 0,Y 425.285,Z 571.508,A -85,B 0,C 180,E1 -9949.478,E2 -9949.478} C_VEL
LIN {X 0,Y 425.279,Z 571.514,A -85,B 0,C 180,E1 -9952.488,E2 -9952.488} C_VEL
LIN {X 0,Y 425.308,Z 571.506,A -85,B 0,C 180,E1 -9955.817,E2 -9955.817} C_VEL
LIN {X 0,Y 425.291,Z 571.509,A -85,B 0,C 180,E1 -9959.238,E2 -9959.238} C_VEL
LIN {X 0,Y 425.349,Z 571.504,A -85,B 0,C 180,E1 -9962.442,E2 -9962.442} C_VEL
LIN {X 0,Y 425.352,Z 571.5,A -85,B 0,C 180,E1 -9965.601,E2 -9965.601} C_VEL
LIN {X 0,Y 425.294,Z 571.512,A -85,B 0,C 180,E1 -9968.681,E2 -9968.681} C_VEL
LIN {X 0,Y 425.333,Z 571.503,A -85,B 0,C 180,E1 -9971.702,E2 -9971.702} C_VEL
LIN {X 0,Y 425.348,Z 571.505,A -85,B 0,C 180,E1 -9974.67,E2 -9974.67} C_VEL
LIN {X 0,Y 425.43,Z 571.49,A -85,B 0,C 180,E1 -9977.598,E2 -9977.598} C_VEL
LIN {X 0,Y 425.442,Z 571.489,A -85,B 0,C 180,E1 -9981.449,E2 -9981.449} C_VEL
LIN {X 0,Y 425.554,Z 571.479,A -85,B 0,C 180,E1 -9984.312,E2 -9984.312} C_VEL
LIN {X 0,Y 425.575,Z 571.475,A -85,B 0,C 180,E1 -9988.106,E2 -9988.106} C_VEL
LIN {X 0,Y 429.061,Z 583.933,A -85,B 0,C 180,E1 -9988.955,E2 -9988.955} C_VEL
LIN {X 0,Y 428.85,Z 595.104,A -85,B 0,C 180,E1 -9989.788,E2 -9989.788} C_VEL
LIN {X 0,Y 428.246,Z 606.222,A -85,B 0,C 180,E1 -9990.822,E2 -9990.822} C_VEL
LIN {X 0,Y 427.723,Z 615.808,A -85,B 0,C 180,E1 -9991.935,E2 -9991.935} C_VEL
LIN {X 0,Y 427.178,Z 623.82,A -85,B 0,C 180,E1 -9993.064,E2 -9993.064} C_VEL
LIN {X 0,Y 426.67,Z 631.985,A -85,B 0,C 180,E1 -9994.487,E2 -9994.487} C_VEL
LIN {X 0,Y 426.498,Z 635.132,A -85,B 0,C 180,E1 -9995.13,E2 -9995.13} C_VEL
LIN {X 0,Y 425.656,Z 638.237,A -85,B 0,C 180,E1 -9995.798,E2 -9995.798} C_VEL
LIN {X 0,Y 422.541,Z 643.004,A -85,B 0,C 180,E1 -9996.895,E2 -9996.895} C_VEL
LIN {X 0,Y 419.42,Z 647.107,A -85,B 0,C 180,E1 -9998.05,E2 -9998.05} C_VEL
LIN {X 0,Y 418.585,Z 649.138,A -85,B 0,C 180,E1 -9998.801,E2 -9998.801} C_VEL
LIN {X 0,Y 418.415,Z 651.091,A -85,B 0,C 180,E1 -9999.669,E2 -9999.669} C_VEL
LIN {X 0,Y 418.288,Z 652.814,A -85,B 0,C 180,E1 -10000.65,E2 -10000.65} C_VEL
LIN {X 0,Y 418.222,Z 655.048,A -85,B 0,C 180,E1 -10002.617,E2 -10002.617} C_VEL
LIN {X 0,Y 418.184,Z 655.549,A -85,B 0,C 180,E1 -10003.607,E2 -10003.607} C_VEL
LIN {X 0,Y 418.21,Z 655.332,A -85,B 0,C 180,E1 -10005.597,E2 -10005.597} C_VEL
LIN {X 0,Y 418.325,Z 654.462,A -85,B 0,C 180,E1 -10006.742,E2 -10006.742} C_VEL
LIN {X 0,Y 418.601,Z 651.845,A -85,B 0,C 180,E1 -10008.601,E2 -10008.601} C_VEL
LIN {X 0,Y 418.971,Z 648.702,A -85,B 0,C 180,E1 -10010.056,E2 -10010.056} C_VEL
LIN {X 0,Y 419.396,Z 644.134,A -85,B 0,C 180,E1 -10011.632,E2 -10011.632} C_VEL
LIN {X 0,Y 419.977,Z 638.169,A -85,B 0,C 180,E1 -10013.207,E2 -10013.207} C_VEL
LIN {X 0,Y 420.592,Z 631.017,A -85,B 0,C 180,E1 -10014.691,E2 -10014.691} C_VEL
LIN {X 0,Y 421.237,Z 623.395,A -85,B 0,C 180,E1 -10015.973,E2 -10015.973} C_VEL
LIN {X 0,Y 421.992,Z 614.023,A -85,B 0,C 180,E1 -10017.257,E2 -10017.257} C_VEL
LIN {X 0,Y 422.647,Z 603.583,A -85,B 0,C 180,E1 -10018.403,E2 -10018.403} C_VEL
LIN {X 0,Y 423.39,Z 592.224,A -85,B 0,C 180,E1 -10019.386,E2 -10019.386} C_VEL
LIN {X 0,Y 423.399,Z 588.262,A -85,B 0,C 180,E1 -10019.687,E2 -10019.687} C_VEL
LIN {X 0,Y 419.863,Z 577.189,A -85,B 0,C 180,E1 -10020.594,E2 -10020.594} C_VEL
LIN {X 0,Y 418.261,Z 572.381,A -85,B 0,C 180,E1 -10020.939,E2 -10020.939} C_VEL
LIN {X 0,Y 418.242,Z 572.385,A -85,B 0,C 180,E1 -10023.676,E2 -10023.676} C_VEL
LIN {X 0,Y 418.243,Z 572.389,A -85,B 0,C 180,E1 -10027.222,E2 -10027.222} C_VEL
LIN {X 0,Y 418.291,Z 572.47,A -85,B 0,C 180,E1 -10028.436,E2 -10028.436} C_VEL
LIN {X 0,Y 419.171,Z 578.147,A -85,B 0,C 180,E1 -10030.834,E2 -10030.834} C_VEL
LIN {X 0,Y 419.29,Z 583.311,A -85,B 0,C 180,E1 -10032.902,E2 -10032.902} C_VEL
LIN {X 0,Y 419.171,Z 591.449,A -85,B 0,C 180,E1 -10036.132,E2 -10036.132} C_VEL
LIN {X 0,Y 418.888,Z 598.99,A -85,B 0,C 180,E1 -10039.132,E2 -10039.132} C_VEL
LIN {X 0,Y 418.73,Z 606.372,A -85,B 0,C 180,E1 -10042.076,E2 -10042.076} C_VEL
LIN {X 0,Y 418.506,Z 615.848,A -85,B 0,C 180,E1 -10045.859,E2 -10045.859} C_VEL
LIN {X 0,Y 418.199,Z 625.613,A -85,B 0,C 180,E1 -10049.725,E2 -10049.725} C_VEL
LIN {X 0,Y 418.171,Z 626.246,A -85,B 0,C 180,E1 -10049.975,E2 -10049.975} C_VEL
LIN {X 0,Y 421.207,Z 641.031,A -85,B 0,C 180,E1 -10050.576,E2 -10050.576} C_VEL
LIN {X 0,Y 422.018,Z 646.824,A -85,B 0,C 180,E1 -10050.864,E2 -10050.864} C_VEL
LIN {X 0,Y 421.507,Z 658.481,A -85,B 0,C 180,E1 -10051.493,E2 -10051.493} C_VEL
LIN {X 0,Y 420.87,Z 671.109,A -85,B 0,C 180,E1 -10052.396,E2 -10052.396} C_VEL
LIN {X 0,Y 420.125,Z 682.378,A -85,B 0,C 180,E1 -10053.418,E2 -10053.418} C_VEL
LIN {X 0,Y 419.502,Z 692.393,A -85,B 0,C 180,E1 -10054.558,E2 -10054.558} C_VEL
LIN {X 0,Y 418.811,Z 702.579,A -85,B 0,C 180,E1 -10055.988,E2 -10055.988} C_VEL
LIN {X 0,Y 418.203,Z 711.39,A -85,B 0,C 180,E1 -10057.558,E2 -10057.558} C_VEL
LIN {X 0,Y 417.824,Z 718.102,A -85,B 0,C 180,E1 -10059.058,E2 -10059.058} C_VEL
LIN {X 0,Y 417.542,Z 723.166,A -85,B 0,C 180,E1 -10060.486,E2 -10060.486} C_VEL
LIN {X 0,Y 417.323,Z 726.948,A -85,B 0,C 180,E1 -10061.848,E2 -10061.848} C_VEL
LIN {X 0,Y 417.129,Z 730.763,A -85,B 0,C 180,E1 -10063.81,E2 -10063.81} C_VEL
LIN {X 0,Y 417.003,Z 732.554,A -85,B 0,C 180,E1 -10065.357,E2 -10065.357} C_VEL
LIN {X 0,Y 417.003,Z 733.165,A -85,B 0,C 180,E1 -10066.353,E2 -10066.353} C_VEL
LIN {X 0,Y 417.096,Z 733.254,A -85,B 0,C 180,E1 -10067.76,E2 -10067.76} C_VEL
LIN {X 0,Y 417.11,Z 732.372,A -85,B 0,C 180,E1 -10069.319,E2 -10069.319} C_VEL
LIN {X 0,Y 417.161,Z 731.252,A -85,B 0,C 180,E1 -10070.301,E2 -10070.301} C_VEL
LIN {X 0,Y 417.27,Z 729.706,A -85,B 0,C 180,E1 -10071.282,E2 -10071.282} C_VEL
LIN {X 0,Y 417.502,Z 726.445,A -85,B 0,C 180,E1 -10072.796,E2 -10072.796} C_VEL
LIN {X 0,Y 417.705,Z 722.369,A -85,B 0,C 180,E1 -10074.206,E2 -10074.206} C_VEL
LIN {X 0,Y 418.059,Z 716.988,A -85,B 0,C 180,E1 -10075.662,E2 -10075.662} C_VEL
LIN {X 0,Y 418.536,Z 710.258,A -85,B 0,C 180,E1 -10077.113,E2 -10077.113} C_VEL
LIN {X 0,Y 419.199,Z 701.84,A -85,B 0,C 180,E1 -10078.559,E2 -10078.559} C_VEL
LIN {X 0,Y 419.866,Z 693.266,A -85,B 0,C 180,E1 -10079.761,E2 -10079.761} C_VEL
LIN {X 0,Y 420.641,Z 682.794,A -85,B 0,C 180,E1 -10080.958,E2 -10080.958} C_VEL
LIN {X 0,Y 421.482,Z 670.951,A -85,B 0,C 180,E1 -10082.031,E2 -10082.031} C_VEL
LIN {X 0,Y 422.118,Z 659.259,A -85,B 0,C 180,E1 -10082.863,E2 -10082.863} C_VEL
LIN {X 0,Y 422.683,Z 646.267,A -85,B 0,C 180,E1 -10083.561,E2 -10083.561} C_VEL
LIN {X 0,Y 419.773,Z 633.455,A -85,B 0,C 180,E1 -10084.216,E2 -10084.216} C_VEL
LIN {X 0,Y 418.529,Z 628.235,A -85,B 0,C 180,E1 -10084.455,E2 -10084.455} C_VEL
LIN {X 0,Y 418.779,Z 619.953,A -85,B 0,C 180,E1 -10087.716,E2 -10087.716} C_VEL
LIN {X 0,Y 419.026,Z 612.499,A -85,B 0,C 180,E1 -10090.632,E2 -10090.632} C_VEL
LIN {X 0,Y 419.278,Z 603.656,A -85,B 0,C 180,E1 -10094.067,E2 -10094.067} C_VEL
LIN {X 0,Y 419.512,Z 594.422,A -85,B 0,C 180,E1 -10097.551,E2 -10097.551} C_VEL
LIN {X 0,Y 419.671,Z 584.673,A -85,B 0,C 180,E1 -10101.104,E2 -10101.104} C_VEL
LIN {X 0,Y 419.543,Z 578.875,A -85,B 0,C 180,E1 -10103.219,E2 -10103.219} C_VEL
LIN {X 0,Y 418.261,Z 572.391,A -85,B 0,C 180,E1 -10105.704,E2 -10105.704} C_VEL
LIN {X 0,Y 418.289,Z 572.383,A -85,B 0,C 180,E1 -10108.064,E2 -10108.064} C_VEL
LIN {X 0,Y 418.211,Z 572.393,A -85,B 0,C 180,E1 -10111.397,E2 -10111.397} C_VEL
LIN {X 0,Y 418.261,Z 572.388,A -85,B 0,C 180,E1 -10114.581,E2 -10114.581} C_VEL
LIN {X 0,Y 418.233,Z 572.391,A -85,B 0,C 180,E1 -10117.836,E2 -10117.836} C_VEL
LIN {X 0,Y 418.263,Z 572.387,A -85,B 0,C 180,E1 -10120.944,E2 -10120.944} C_VEL
LIN {X 0,Y 418.28,Z 572.384,A -85,B 0,C 180,E1 -10123.741,E2 -10123.741} C_VEL
LIN {X 0,Y 418.311,Z 572.577,A -85,B 0,C 180,E1 -10126.533,E2 -10126.533} C_VEL
LIN {X 0,Y 420.149,Z 581.342,A -85,B 0,C 180,E1 -10129.675,E2 -10129.675} C_VEL
LIN {X 0,Y 421.765,Z 589.929,A -85,B 0,C 180,E1 -10132.542,E2 -10132.542} C_VEL
LIN {X 0,Y 421.797,Z 593.829,A -85,B 0,C 180,E1 -10133.738,E2 -10133.738} C_VEL
LIN {X 0,Y 420.974,Z 603.601,A -85,B 0,C 180,E1 -10136.588,E2 -10136.588} C_VEL
LIN {X 0,Y 420.078,Z 616.558,A -85,B 0,C 180,E1 -10140.23,E2 -10140.23} C_VEL
LIN {X 0,Y 419.304,Z 629.097,A -85,B 0,C 180,E1 -10143.631,E2 -10143.631} C_VEL
LIN {X 0,Y 418.714,Z 640.967,A -85,B 0,C 180,E1 -10146.77,E2 -10146.77} C_VEL
LIN {X 0,Y 418.196,Z 654.359,A -85,B 0,C 180,E1 -10150.239,E2 -10150.239} C_VEL
LIN {X 0,Y 417.967,Z 663.161,A -85,B 0,C 180,E1 -10152.501,E2 -10152.501} C_VEL
LIN {X 0,Y 419.711,Z 677.863,A -85,B 0,C 180,E1 -10152.992,E2 -10152.992} C_VEL
LIN {X 0,Y 420.462,Z 690.224,A -85,B 0,C 180,E1 -10153.555,E2 -10153.555} C_VEL
LIN {X 0,Y 421.2,Z 700.73,A -85,B 0,C 180,E1 -10154.145,E2 -10154.145} C_VEL
LIN {X 0,Y 420.481,Z 713.869,A -85,B 0,C 180,E1 -10154.986,E2 -10154.986} C_VEL
LIN {X 0,Y 419.729,Z 725.469,A -85,B 0,C 180,E1 -10155.95,E2 -10155.95} C_VEL
LIN {X 0,Y 419.147,Z 735.242,A -85,B 0,C 180,E1 -10156.956,E2 -10156.956} C_VEL
LIN {X 0,Y 418.548,Z 744.644,A -85,B 0,C 180,E1 -10158.131,E2 -10158.131} C_VEL
LIN {X 0,Y 418.014,Z 752.648,A -85,B 0,C 180,E1 -10159.343,E2 -10159.343} C_VEL
LIN {X 0,Y 417.661,Z 760.476,A -85,B 0,C 180,E1 -10160.802,E2 -10160.802} C_VEL
LIN {X 0,Y 417.401,Z 766.78,A -85,B 0,C 180,E1 -10162.26,E2 -10162.26} C_VEL
LIN {X 0,Y 417.258,Z 771.412,A -85,B 0,C 180,E1 -10163.596,E2 -10163.596} C_VEL
LIN {X 0,Y 417.255,Z 775.616,A -85,B 0,C 180,E1 -10165.17,E2 -10165.17} C_VEL
LIN {X 0,Y 417.185,Z 777.597,A -85,B 0,C 180,E1 -10166.137,E2 -10166.137} C_VEL
LIN {X 0,Y 417.261,Z 779.093,A -85,B 0,C 180,E1 -10167.105,E2 -10167.105} C_VEL
LIN {X 0,Y 417.239,Z 780.161,A -85,B 0,C 180,E1 -10168.07,E2 -10168.07} C_VEL
LIN {X 0,Y 417.261,Z 780.823,A -85,B 0,C 180,E1 -10169.036,E2 -10169.036} C_VEL
LIN {X 0,Y 417.256,Z 781.049,A -85,B 0,C 180,E1 -10170.001,E2 -10170.001} C_VEL
LIN {X 0,Y 417.277,Z 780.828,A -85,B 0,C 180,E1 -10170.966,E2 -10170.966} C_VEL
LIN {X 0,Y 417.24,Z 780.201,A -85,B 0,C 180,E1 -10171.931,E2 -10171.931} C_VEL
LIN {X 0,Y 417.258,Z 779.166,A -85,B 0,C 180,E1 -10172.897,E2 -10172.897} C_VEL
LIN {X 0,Y 417.172,Z 777.647,A -85,B 0,C 180,E1 -10173.865,E2 -10173.865} C_VEL
LIN {X 0,Y 417.279,Z 774.553,A -85,B 0,C 180,E1 -10175.316,E2 -10175.316} C_VEL
LIN {X 0,Y 417.273,Z 770.337,A -85,B 0,C 180,E1 -10176.772,E2 -10176.772} C_VEL
LIN {X 0,Y 417.537,Z 763.885,A -85,B 0,C 180,E1 -10178.47,E2 -10178.47} C_VEL
LIN {X 0,Y 417.847,Z 756.781,A -85,B 0,C 180,E1 -10179.928,E2 -10179.928} C_VEL
LIN {X 0,Y 418.338,Z 747.878,A -85,B 0,C 180,E1 -10181.386,E2 -10181.386} C_VEL
LIN {X 0,Y 418.874,Z 738.747,A -85,B 0,C 180,E1 -10182.599,E2 -10182.599} C_VEL
LIN {X 0,Y 419.421,Z 728.856,A -85,B 0,C 180,E1 -10183.668,E2 -10183.668} C_VEL
LIN {X 0,Y 420.143,Z 717.432,A -85,B 0,C 180,E1 -10184.656,E2 -10184.656} C_VEL
LIN {X 0,Y 420.813,Z 705.935,A -85,B 0,C 180,E1 -10185.437,E2 -10185.437} C_VEL
LIN {X 0,Y 420.939,Z 698.095,A -85,B 0,C 180,E1 -10185.867,E2 -10185.867} C_VEL
LIN {X 0,Y 420.044,Z 688.247,A -85,B 0,C 180,E1 -10186.339,E2 -10186.339} C_VEL
LIN {X 0,Y 418.856,Z 673.55,A -85,B 0,C 180,E1 -10186.916,E2 -10186.916} C_VEL
LIN {X 0,Y 417.926,Z 664.093,A -85,B 0,C 180,E1 -10187.189,E2 -10187.189} C_VEL
LIN {X 0,Y 418.252,Z 652.444,A -85,B 0,C 180,E1 -10190.155,E2 -10190.155} C_VEL
LIN {X 0,Y 418.755,Z 638.397,A -85,B 0,C 180,E1 -10193.754,E2 -10193.754} C_VEL
LIN {X 0,Y 419.41,Z 624.54,A -85,B 0,C 180,E1 -10197.362,E2 -10197.362} C_VEL
LIN {X 0,Y 420.129,Z 611.018,A -85,B 0,C 180,E1 -10200.958,E2 -10200.958} C_VEL
LIN {X 0,Y 420.882,Z 598.758,A -85,B 0,C 180,E1 -10204.304,E2 -10204.304} C_VEL
LIN {X 0,Y 421.377,Z 589.487,A -85,B 0,C 180,E1 -10206.902,E2 -10206.902} C_VEL
LIN {X 0,Y 420.142,Z 582.059,A -85,B 0,C 180,E1 -10209.159,E2 -10209.159} C_VEL
LIN {X 0,Y 418.269,Z 572.386,A -85,B 0,C 180,E1 -10212.278,E2 -10212.278} C_VEL
LIN {X 0,Y 418.241,Z 572.389,A -85,B 0,C 180,E1 -10215.109,E2 -10215.109} C_VEL
LIN {X 0,Y 418.245,Z 572.388,A -85,B 0,C 180,E1 -10217.767,E2 -10217.767} C_VEL
LIN {X 0,Y 418.265,Z 572.385,A -85,B 0,C 180,E1 -10220.618,E2 -10220.618} C_VEL
LIN {X 0,Y 418.251,Z 572.388,A -85,B 0,C 180,E1 -10223.976,E2 -10223.976} C_VEL
LIN {X 0,Y 418.262,Z 572.383,A -85,B 0,C 180,E1 -10227.156,E2 -10227.156} C_VEL
LIN {X 0,Y 418.273,Z 572.382,A -85,B 0,C 180,E1 -10230.895,E2 -10230.895} C_VEL
LIN {X 0,Y 418.276,Z 572.385,A -85,B 0,C 180,E1 -10234.096,E2 -10234.096} C_VEL
LIN {X 0,Y 418.243,Z 572.385,A -85,B 0,C 180,E1 -10237.264,E2 -10237.264} C_VEL
LIN {X 0,Y 418.288,Z 572.384,A -85,B 0,C 180,E1 -10240.364,E2 -10240.364} C_VEL
LIN {X 0,Y 418.322,Z 572.376,A -85,B 0,C 180,E1 -10243.404,E2 -10243.404} C_VEL
LIN {X 0,Y 418.351,Z 572.373,A -85,B 0,C 180,E1 -10246.999,E2 -10246.999} C_VEL
LIN {X 0,Y 418.345,Z 572.377,A -85,B 0,C 180,E1 -10250.328,E2 -10250.328} C_VEL
LIN {X 0,Y 418.518,Z 572.355,A -85,B 0,C 180,E1 -10252.279,E2 -10252.279} C_VEL
LIN {X 0,Y 418.517,Z 572.355,A -85,B 0,C 180,E1 -10254.217,E2 -10254.217} C_VEL
LIN {X 0,Y 418.546,Z 572.352,A -85,B 0,C 180,E1 -10258.075,E2 -10258.075} C_VEL
LIN {X 0,Y 418.677,Z 572.334,A -85,B 0,C 180,E1 -10260,E2 -10260} C_VEL
LIN {X 0,Y 418.504,Z 572.355,A -85,B 0,C 180,E1 -10262.887,E2 -10262.887} C_VEL
LIN {X 0,Y 418.498,Z 572.357,A -85,B 0,C 180,E1 -10266.751,E2 -10266.751} C_VEL
LIN {X 0,Y 418.404,Z 572.369,A -85,B 0,C 180,E1 -10268.695,E2 -10268.695} C_VEL
LIN {X 0,Y 418.318,Z 572.376,A -85,B 0,C 180,E1 -10271.631,E2 -10271.631} C_VEL
LIN {X 0,Y 418.306,Z 572.381,A -85,B 0,C 180,E1 -10274.596,E2 -10274.596} C_VEL
LIN {X 0,Y 418.291,Z 572.38,A -85,B 0,C 180,E1 -10277.603,E2 -10277.603} C_VEL
LIN {X 0,Y 418.253,Z 572.388,A -85,B 0,C 180,E1 -10280.662,E2 -10280.662} C_VEL
LIN {X 0,Y 418.291,Z 572.381,A -85,B 0,C 180,E1 -10283.781,E2 -10283.781} C_VEL
LIN {X 0,Y 418.312,Z 572.377,A -85,B 0,C 180,E1 -10287.07,E2 -10287.07} C_VEL
LIN {X 0,Y 418.246,Z 572.389,A -85,B 0,C 180,E1 -10290.271,E2 -10290.271} C_VEL
LIN {X 0,Y 418.251,Z 572.385,A -85,B 0,C 180,E1 -10293.676,E2 -10293.676} C_VEL
LIN {X 0,Y 418.247,Z 572.386,A -85,B 0,C 180,E1 -10297.223,E2 -10297.223} C_VEL
LIN {X 0,Y 418.252,Z 572.385,A -85,B 0,C 180,E1 -10299.681,E2 -10299.681} C_VEL
LIN {X 0,Y 418.234,Z 572.391,A -85,B 0,C 180,E1 -10302.321,E2 -10302.321} C_VEL
LIN {X 0,Y 418.243,Z 572.387,A -85,B 0,C 180,E1 -10305.109,E2 -10305.109} C_VEL
LIN {X 0,Y 418.244,Z 572.386,A -85,B 0,C 180,E1 -10307.766,E2 -10307.766} C_VEL
LIN {X 0,Y 418.259,Z 572.387,A -85,B 0,C 180,E1 -10310.618,E2 -10310.618} C_VEL
LIN {X 0,Y 418.243,Z 572.387,A -85,B 0,C 180,E1 -10313.975,E2 -10313.975} C_VEL
LIN {X 0,Y 418.258,Z 572.385,A -85,B 0,C 180,E1 -10317.155,E2 -10317.155} C_VEL
LIN {X 0,Y 418.269,Z 572.385,A -85,B 0,C 180,E1 -10320.895,E2 -10320.895} C_VEL
LIN {X 0,Y 418.271,Z 572.384,A -85,B 0,C 180,E1 -10324.095,E2 -10324.095} C_VEL
LIN {X 0,Y 418.238,Z 572.387,A -85,B 0,C 180,E1 -10327.263,E2 -10327.263} C_VEL
LIN {X 0,Y 418.283,Z 572.385,A -85,B 0,C 180,E1 -10330.363,E2 -10330.363} C_VEL
LIN {X 0,Y 418.317,Z 572.377,A -85,B 0,C 180,E1 -10333.404,E2 -10333.404} C_VEL
LIN {X 0,Y 418.355,Z 572.374,A -85,B 0,C 180,E1 -10336.993,E2 -10336.993} C_VEL
LIN {X 0,Y 418.359,Z 572.374,A -85,B 0,C 180,E1 -10340.328,E2 -10340.328} C_VEL
LIN {X 0,Y 418.493,Z 572.355,A -85,B 0,C 180,E1 -10343.248,E2 -10343.248} C_VEL
LIN {X 0,Y 418.341,Z 572.375,A -85,B 0,C 180,E1 -10345.181,E2 -10345.181} C_VEL
LIN {X 0,Y 418.519,Z 572.355,A -85,B 0,C 180,E1 -10347.864,E2 -10347.864} C_VEL
LIN {X 0,Y 421.99,Z 584.598,A -85,B 0,C 180,E1 -10348.712,E2 -10348.712} C_VEL
LIN {X 0,Y 422.284,Z 587.823,A -85,B 0,C 180,E1 -10348.95,E2 -10348.95} C_VEL
LIN {X 0,Y 421.799,Z 599.156,A -85,B 0,C 180,E1 -10349.849,E2 -10349.849} C_VEL
LIN {X 0,Y 421.187,Z 610.094,A -85,B 0,C 180,E1 -10350.955,E2 -10350.955} C_VEL
LIN {X 0,Y 420.647,Z 619.625,A -85,B 0,C 180,E1 -10352.153,E2 -10352.153} C_VEL
LIN {X 0,Y 420.06,Z 627.485,A -85,B 0,C 180,E1 -10353.356,E2 -10353.356} C_VEL
LIN {X 0,Y 419.605,Z 635.156,A -85,B 0,C 180,E1 -10354.803,E2 -10354.803} C_VEL
LIN {X 0,Y 419.15,Z 641.317,A -85,B 0,C 180,E1 -10356.256,E2 -10356.256} C_VEL
LIN {X 0,Y 418.751,Z 647.129,A -85,B 0,C 180,E1 -10358.026,E2 -10358.026} C_VEL
LIN {X 0,Y 418.585,Z 649.138,A -85,B 0,C 180,E1 -10358.801,E2 -10358.801} C_VEL
LIN {X 0,Y 417.767,Z 650.977,A -85,B 0,C 180,E1 -10359.565,E2 -10359.565} C_VEL
LIN {X 0,Y 414.741,Z 653.619,A -85,B 0,C 180,E1 -10360.813,E2 -10360.813} C_VEL
LIN {X 0,Y 411.821,Z 655.573,A -85,B 0,C 180,E1 -10362.098,E2 -10362.098} C_VEL
LIN {X 0,Y 411.181,Z 656.23,A -85,B 0,C 180,E1 -10362.91,E2 -10362.91} C_VEL
LIN {X 0,Y 411.169,Z 656.626,A -85,B 0,C 180,E1 -10364.855,E2 -10364.855} C_VEL
LIN {X 0,Y 411.214,Z 656.255,A -85,B 0,C 180,E1 -10365.869,E2 -10365.869} C_VEL
LIN {X 0,Y 411.344,Z 655.394,A -85,B 0,C 180,E1 -10366.907,E2 -10366.907} C_VEL
LIN {X 0,Y 411.493,Z 654.173,A -85,B 0,C 180,E1 -10367.903,E2 -10367.903} C_VEL
LIN {X 0,Y 411.797,Z 651.468,A -85,B 0,C 180,E1 -10369.438,E2 -10369.438} C_VEL
LIN {X 0,Y 412.216,Z 647.669,A -85,B 0,C 180,E1 -10370.978,E2 -10370.978} C_VEL
LIN {X 0,Y 412.722,Z 642.649,A -85,B 0,C 180,E1 -10372.527,E2 -10372.527} C_VEL
LIN {X 0,Y 413.354,Z 636.198,A -85,B 0,C 180,E1 -10374.082,E2 -10374.082} C_VEL
LIN {X 0,Y 414.091,Z 628.558,A -85,B 0,C 180,E1 -10375.539,E2 -10375.539} C_VEL
LIN {X 0,Y 414.907,Z 619.436,A -85,B 0,C 180,E1 -10376.942,E2 -10376.942} C_VEL
LIN {X 0,Y 415.602,Z 609.942,A -85,B 0,C 180,E1 -10378.122,E2 -10378.122} C_VEL
LIN {X 0,Y 416.316,Z 599.431,A -85,B 0,C 180,E1 -10379.168,E2 -10379.168} C_VEL
LIN {X 0,Y 416.691,Z 590.004,A -85,B 0,C 180,E1 -10379.937,E2 -10379.937} C_VEL
LIN {X 0,Y 412.906,Z 578.212,A -85,B 0,C 180,E1 -10380.935,E2 -10380.935} C_VEL
LIN {X 0,Y 411.187,Z 573.261,A -85,B 0,C 180,E1 -10381.317,E2 -10381.317} C_VEL
LIN {X 0,Y 411.2,Z 573.264,A -85,B 0,C 180,E1 -10384.333,E2 -10384.333} C_VEL
LIN {X 0,Y 411.261,Z 573.357,A -85,B 0,C 180,E1 -10388.231,E2 -10388.231} C_VEL
LIN {X 0,Y 412.105,Z 578.51,A -85,B 0,C 180,E1 -10390.393,E2 -10390.393} C_VEL
LIN {X 0,Y 412.342,Z 583.021,A -85,B 0,C 180,E1 -10392.257,E2 -10392.257} C_VEL
LIN {X 0,Y 412.192,Z 591.694,A -85,B 0,C 180,E1 -10395.733,E2 -10395.733} C_VEL
LIN {X 0,Y 411.926,Z 598.952,A -85,B 0,C 180,E1 -10398.649,E2 -10398.649} C_VEL
LIN {X 0,Y 411.702,Z 607.491,A -85,B 0,C 180,E1 -10402.082,E2 -10402.082} C_VEL
LIN {X 0,Y 411.504,Z 616.507,A -85,B 0,C 180,E1 -10405.695,E2 -10405.695} C_VEL
LIN {X 0,Y 411.181,Z 626.177,A -85,B 0,C 180,E1 -10409.556,E2 -10409.556} C_VEL
LIN {X 0,Y 411.151,Z 626.593,A -85,B 0,C 180,E1 -10409.724,E2 -10409.724} C_VEL
LIN {X 0,Y 413.976,Z 640.249,A -85,B 0,C 180,E1 -10410.279,E2 -10410.279} C_VEL
LIN {X 0,Y 415.119,Z 646.461,A -85,B 0,C 180,E1 -10410.596,E2 -10410.596} C_VEL
LIN {X 0,Y 414.572,Z 659.539,A -85,B 0,C 180,E1 -10411.317,E2 -10411.317} C_VEL
LIN {X 0,Y 413.892,Z 672.464,A -85,B 0,C 180,E1 -10412.272,E2 -10412.272} C_VEL
LIN {X 0,Y 413.124,Z 683.771,A -85,B 0,C 180,E1 -10413.341,E2 -10413.341} C_VEL
LIN {X 0,Y 412.457,Z 694.113,A -85,B 0,C 180,E1 -10414.563,E2 -10414.563} C_VEL
LIN {X 0,Y 411.808,Z 702.83,A -85,B 0,C 180,E1 -10415.821,E2 -10415.821} C_VEL
LIN {X 0,Y 411.192,Z 711.382,A -85,B 0,C 180,E1 -10417.359,E2 -10417.359} C_VEL
LIN {X 0,Y 410.789,Z 718.42,A -85,B 0,C 180,E1 -10418.945,E2 -10418.945} C_VEL
LIN {X 0,Y 410.421,Z 724.315,A -85,B 0,C 180,E1 -10420.671,E2 -10420.671} C_VEL
LIN {X 0,Y 410.168,Z 729.016,A -85,B 0,C 180,E1 -10422.552,E2 -10422.552} C_VEL
LIN {X 0,Y 410.028,Z 731.605,A -85,B 0,C 180,E1 -10424.083,E2 -10424.083} C_VEL
LIN {X 0,Y 409.939,Z 732.734,A -85,B 0,C 180,E1 -10425.099,E2 -10425.099} C_VEL
LIN {X 0,Y 409.921,Z 733.443,A -85,B 0,C 180,E1 -10426.112,E2 -10426.112} C_VEL
LIN {X 0,Y 410.013,Z 733.686,A -85,B 0,C 180,E1 -10427.69,E2 -10427.69} C_VEL
LIN {X 0,Y 410.029,Z 732.991,A -85,B 0,C 180,E1 -10429.133,E2 -10429.133} C_VEL
LIN {X 0,Y 410.065,Z 732.018,A -85,B 0,C 180,E1 -10430.132,E2 -10430.132} C_VEL
LIN {X 0,Y 410.182,Z 730.58,A -85,B 0,C 180,E1 -10431.13,E2 -10431.13} C_VEL
LIN {X 0,Y 410.42,Z 727.61,A -85,B 0,C 180,E1 -10432.622,E2 -10432.622} C_VEL
LIN {X 0,Y 410.63,Z 723.597,A -85,B 0,C 180,E1 -10434.106,E2 -10434.106} C_VEL
LIN {X 0,Y 410.99,Z 718.408,A -85,B 0,C 180,E1 -10435.587,E2 -10435.587} C_VEL
LIN {X 0,Y 411.482,Z 711.924,A -85,B 0,C 180,E1 -10437.063,E2 -10437.063} C_VEL
LIN {X 0,Y 412.164,Z 703.89,A -85,B 0,C 180,E1 -10438.535,E2 -10438.535} C_VEL
LIN {X 0,Y 413.017,Z 693.808,A -85,B 0,C 180,E1 -10440,E2 -10440} C_VEL
LIN {X 0,Y 413.816,Z 683.37,A -85,B 0,C 180,E1 -10441.217,E2 -10441.217} C_VEL
LIN {X 0,Y 414.708,Z 671.555,A -85,B 0,C 180,E1 -10442.307,E2 -10442.307} C_VEL
LIN {X 0,Y 415.391,Z 659.92,A -85,B 0,C 180,E1 -10443.152,E2 -10443.152} C_VEL
LIN {X 0,Y 416.026,Z 647.929,A -85,B 0,C 180,E1 -10443.814,E2 -10443.814} C_VEL
LIN {X 0,Y 413.033,Z 634.421,A -85,B 0,C 180,E1 -10444.545,E2 -10444.545} C_VEL
LIN {X 0,Y 411.521,Z 628.701,A -85,B 0,C 180,E1 -10444.831,E2 -10444.831} C_VEL
LIN {X 0,Y 411.842,Z 621.093,A -85,B 0,C 180,E1 -10447.847,E2 -10447.847} C_VEL
LIN {X 0,Y 412.085,Z 613.566,A -85,B 0,C 180,E1 -10450.813,E2 -10450.813} C_VEL
LIN {X 0,Y 412.367,Z 604.678,A -85,B 0,C 180,E1 -10454.308,E2 -10454.308} C_VEL
LIN {X 0,Y 412.573,Z 598.11,A -85,B 0,C 180,E1 -10456.834,E2 -10456.834} C_VEL
LIN {X 0,Y 412.753,Z 589.854,A -85,B 0,C 180,E1 -10459.91,E2 -10459.91} C_VEL
LIN {X 0,Y 412.848,Z 582.821,A -85,B 0,C 180,E1 -10462.521,E2 -10462.521} C_VEL
LIN {X 0,Y 412.344,Z 578.575,A -85,B 0,C 180,E1 -10464.146,E2 -10464.146} C_VEL
LIN {X 0,Y 411.229,Z 573.266,A -85,B 0,C 180,E1 -10466.245,E2 -10466.245} C_VEL
LIN {X 0,Y 411.235,Z 573.262,A -85,B 0,C 180,E1 -10469.359,E2 -10469.359} C_VEL
LIN {X 0,Y 411.201,Z 573.267,A -85,B 0,C 180,E1 -10473.157,E2 -10473.157} C_VEL
LIN {X 0,Y 411.191,Z 573.266,A -85,B 0,C 180,E1 -10476.554,E2 -10476.554} C_VEL
LIN {X 0,Y 411.223,Z 573.262,A -85,B 0,C 180,E1 -10479.731,E2 -10479.731} C_VEL
LIN {X 0,Y 411.227,Z 573.262,A -85,B 0,C 180,E1 -10483.127,E2 -10483.127} C_VEL
LIN {X 0,Y 411.249,Z 573.444,A -85,B 0,C 180,E1 -10486.096,E2 -10486.096} C_VEL
LIN {X 0,Y 412.985,Z 581.732,A -85,B 0,C 180,E1 -10489.147,E2 -10489.147} C_VEL
LIN {X 0,Y 414.543,Z 589.631,A -85,B 0,C 180,E1 -10491.864,E2 -10491.864} C_VEL
LIN {X 0,Y 414.955,Z 593.73,A -85,B 0,C 180,E1 -10493.203,E2 -10493.203} C_VEL
LIN {X 0,Y 414.17,Z 602.91,A -85,B 0,C 180,E1 -10495.947,E2 -10495.947} C_VEL
LIN {X 0,Y 413.248,Z 614.602,A -85,B 0,C 180,E1 -10499.324,E2 -10499.324} C_VEL
LIN {X 0,Y 412.496,Z 626.365,A -85,B 0,C 180,E1 -10502.613,E2 -10502.613} C_VEL
LIN {X 0,Y 411.805,Z 638.174,A -85,B 0,C 180,E1 -10505.822,E2 -10505.822} C_VEL
LIN {X 0,Y 411.214,Z 651.956,A -85,B 0,C 180,E1 -10509.492,E2 -10509.492} C_VEL
LIN {X 0,Y 410.899,Z 662.031,A -85,B 0,C 180,E1 -10512.133,E2 -10512.133} C_VEL
LIN {X 0,Y 412.883,Z 677.834,A -85,B 0,C 180,E1 -10512.699,E2 -10512.699} C_VEL
LIN {X 0,Y 414.064,Z 696.593,A -85,B 0,C 180,E1 -10513.611,E2 -10513.611} C_VEL
LIN {X 0,Y 414.292,Z 703.129,A -85,B 0,C 180,E1 -10514,E2 -10514} C_VEL
LIN {X 0,Y 413.541,Z 715.474,A -85,B 0,C 180,E1 -10514.854,E2 -10514.854} C_VEL
LIN {X 0,Y 412.734,Z 726.627,A -85,B 0,C 180,E1 -10515.832,E2 -10515.832} C_VEL
LIN {X 0,Y 412.043,Z 737.17,A -85,B 0,C 180,E1 -10516.984,E2 -10516.984} C_VEL
LIN {X 0,Y 411.447,Z 746.055,A -85,B 0,C 180,E1 -10518.173,E2 -10518.173} C_VEL
LIN {X 0,Y 410.839,Z 755.12,A -85,B 0,C 180,E1 -10519.654,E2 -10519.654} C_VEL
LIN {X 0,Y 410.538,Z 762.42,A -85,B 0,C 180,E1 -10521.138,E2 -10521.138} C_VEL
LIN {X 0,Y 410.287,Z 768.241,A -85,B 0,C 180,E1 -10522.62,E2 -10522.62} C_VEL
LIN {X 0,Y 410.154,Z 772.818,A -85,B 0,C 180,E1 -10524.1,E2 -10524.1} C_VEL
LIN {X 0,Y 410.183,Z 775.243,A -85,B 0,C 180,E1 -10525.086,E2 -10525.086} C_VEL
LIN {X 0,Y 410.094,Z 777.214,A -85,B 0,C 180,E1 -10526.07,E2 -10526.07} C_VEL
LIN {X 0,Y 410.171,Z 778.7,A -85,B 0,C 180,E1 -10527.054,E2 -10527.054} C_VEL
LIN {X 0,Y 410.16,Z 779.763,A -85,B 0,C 180,E1 -10528.037,E2 -10528.037} C_VEL
LIN {X 0,Y 410.172,Z 780.42,A -85,B 0,C 180,E1 -10529.019,E2 -10529.019} C_VEL
LIN {X 0,Y 410.196,Z 780.636,A -85,B 0,C 180,E1 -10530.001,E2 -10530.001} C_VEL
LIN {X 0,Y 410.187,Z 780.41,A -85,B 0,C 180,E1 -10530.983,E2 -10530.983} C_VEL
LIN {X 0,Y 410.161,Z 779.777,A -85,B 0,C 180,E1 -10531.965,E2 -10531.965} C_VEL
LIN {X 0,Y 410.168,Z 778.731,A -85,B 0,C 180,E1 -10532.947,E2 -10532.947} C_VEL
LIN {X 0,Y 410.083,Z 777.198,A -85,B 0,C 180,E1 -10533.932,E2 -10533.932} C_VEL
LIN {X 0,Y 410.186,Z 774.084,A -85,B 0,C 180,E1 -10535.408,E2 -10535.408} C_VEL
LIN {X 0,Y 410.196,Z 769.846,A -85,B 0,C 180,E1 -10536.889,E2 -10536.889} C_VEL
LIN {X 0,Y 410.483,Z 763.369,A -85,B 0,C 180,E1 -10538.617,E2 -10538.617} C_VEL
LIN {X 0,Y 410.784,Z 756.22,A -85,B 0,C 180,E1 -10540.101,E2 -10540.101} C_VEL
LIN {X 0,Y 411.313,Z 747.285,A -85,B 0,C 180,E1 -10541.583,E2 -10541.583} C_VEL
LIN {X 0,Y 411.925,Z 738.114,A -85,B 0,C 180,E1 -10542.815,E2 -10542.815} C_VEL
LIN {X 0,Y 412.51,Z 727.912,A -85,B 0,C 180,E1 -10543.926,E2 -10543.926} C_VEL
LIN {X 0,Y 413.227,Z 716.669,A -85,B 0,C 180,E1 -10544.907,E2 -10544.907} C_VEL
LIN {X 0,Y 413.923,Z 705.068,A -85,B 0,C 180,E1 -10545.701,E2 -10545.701} C_VEL
LIN {X 0,Y 413.936,Z 698.354,A -85,B 0,C 180,E1 -10546.078,E2 -10546.078} C_VEL
LIN {X 0,Y 413.068,Z 687.803,A -85,B 0,C 180,E1 -10546.586,E2 -10546.586} C_VEL
LIN {X 0,Y 411.545,Z 670.185,A -85,B 0,C 180,E1 -10547.252,E2 -10547.252} C_VEL
LIN {X 0,Y 410.881,Z 663.089,A -85,B 0,C 180,E1 -10547.455,E2 -10547.455} C_VEL
LIN {X 0,Y 411.282,Z 649.358,A -85,B 0,C 180,E1 -10551.03,E2 -10551.03} C_VEL
LIN {X 0,Y 411.82,Z 635.322,A -85,B 0,C 180,E1 -10554.716,E2 -10554.716} C_VEL
LIN {X 0,Y 412.449,Z 622.966,A -85,B 0,C 180,E1 -10557.999,E2 -10557.999} C_VEL
LIN {X 0,Y 413.13,Z 611.115,A -85,B 0,C 180,E1 -10561.225,E2 -10561.225} C_VEL
LIN {X 0,Y 413.959,Z 598.747,A -85,B 0,C 180,E1 -10564.664,E2 -10564.664} C_VEL
LIN {X 0,Y 414.421,Z 591.38,A -85,B 0,C 180,E1 -10566.771,E2 -10566.771} C_VEL
LIN {X 0,Y 413.57,Z 585.44,A -85,B 0,C 180,E1 -10568.583,E2 -10568.583} C_VEL
LIN {X 0,Y 411.695,Z 575.609,A -85,B 0,C 180,E1 -10571.742,E2 -10571.742} C_VEL
LIN {X 0,Y 411.217,Z 573.265,A -85,B 0,C 180,E1 -10572.554,E2 -10572.554} C_VEL
LIN {X 0,Y 411.173,Z 573.269,A -85,B 0,C 180,E1 -10575.881,E2 -10575.881} C_VEL
LIN {X 0,Y 411.169,Z 573.27,A -85,B 0,C 180,E1 -10578.772,E2 -10578.772} C_VEL
LIN {X 0,Y 411.216,Z 573.263,A -85,B 0,C 180,E1 -10581.83,E2 -10581.83} C_VEL
LIN {X 0,Y 411.216,Z 573.261,A -85,B 0,C 180,E1 -10585.121,E2 -10585.121} C_VEL
LIN {X 0,Y 411.17,Z 573.269,A -85,B 0,C 180,E1 -10588.003,E2 -10588.003} C_VEL
LIN {X 0,Y 411.223,Z 573.259,A -85,B 0,C 180,E1 -10591.41,E2 -10591.41} C_VEL
LIN {X 0,Y 411.243,Z 573.258,A -85,B 0,C 180,E1 -10593.619,E2 -10593.619} C_VEL
LIN {X 0,Y 411.208,Z 573.263,A -85,B 0,C 180,E1 -10596.852,E2 -10596.852} C_VEL
LIN {X 0,Y 411.22,Z 573.263,A -85,B 0,C 180,E1 -10600.05,E2 -10600.05} C_VEL
LIN {X 0,Y 411.268,Z 573.254,A -85,B 0,C 180,E1 -10603.131,E2 -10603.131} C_VEL
LIN {X 0,Y 411.31,Z 573.251,A -85,B 0,C 180,E1 -10606.896,E2 -10606.896} C_VEL
LIN {X 0,Y 411.297,Z 573.254,A -85,B 0,C 180,E1 -10610.161,E2 -10610.161} C_VEL
LIN {X 0,Y 411.465,Z 573.23,A -85,B 0,C 180,E1 -10613.133,E2 -10613.133} C_VEL
LIN {X 0,Y 411.313,Z 573.249,A -85,B 0,C 180,E1 -10615.099,E2 -10615.099} C_VEL
LIN {X 0,Y 411.515,Z 573.227,A -85,B 0,C 180,E1 -10618.042,E2 -10618.042} C_VEL
LIN {X 0,Y 411.646,Z 573.209,A -85,B 0,C 180,E1 -10620,E2 -10620} C_VEL
LIN {X 0,Y 411.46,Z 573.232,A -85,B 0,C 180,E1 -10622.937,E2 -10622.937} C_VEL
LIN {X 0,Y 411.464,Z 573.232,A -85,B 0,C 180,E1 -10626.866,E2 -10626.866} C_VEL
LIN {X 0,Y 411.358,Z 573.246,A -85,B 0,C 180,E1 -10628.845,E2 -10628.845} C_VEL
LIN {X 0,Y 411.287,Z 573.253,A -85,B 0,C 180,E1 -10631.832,E2 -10631.832} C_VEL
LIN {X 0,Y 411.263,Z 573.257,A -85,B 0,C 180,E1 -10634.852,E2 -10634.852} C_VEL
LIN {X 0,Y 411.256,Z 573.258,A -85,B 0,C 180,E1 -10637.914,E2 -10637.914} C_VEL
LIN {X 0,Y 411.199,Z 573.264,A -85,B 0,C 180,E1 -10641.034,E2 -10641.034} C_VEL
LIN {X 0,Y 411.23,Z 573.262,A -85,B 0,C 180,E1 -10644.215,E2 -10644.215} C_VEL
LIN {X 0,Y 411.261,Z 573.254,A -85,B 0,C 180,E1 -10647.477,E2 -10647.477} C_VEL
LIN {X 0,Y 411.191,Z 573.267,A -85,B 0,C 180,E1 -10650.847,E2 -10650.847} C_VEL
LIN {X 0,Y 411.208,Z 573.266,A -85,B 0,C 180,E1 -10654.333,E2 -10654.333} C_VEL
LIN {X 0,Y 411.202,Z 573.264,A -85,B 0,C 180,E1 -10657.972,E2 -10657.972} C_VEL
LIN {X 0,Y 411.165,Z 573.267,A -85,B 0,C 180,E1 -10661.228,E2 -10661.228} C_VEL
LIN {X 0,Y 411.182,Z 573.269,A -85,B 0,C 180,E1 -10664.489,E2 -10664.489} C_VEL
LIN {X 0,Y 411.18,Z 573.269,A -85,B 0,C 180,E1 -10668.194,E2 -10668.194} C_VEL
LIN {X 0,Y 411.223,Z 573.263,A -85,B 0,C 180,E1 -10670.776,E2 -10670.776} C_VEL
LIN {X 0,Y 411.198,Z 573.267,A -85,B 0,C 180,E1 -10674.47,E2 -10674.47} C_VEL
LIN {X 0,Y 411.208,Z 573.265,A -85,B 0,C 180,E1 -10676.873,E2 -10676.873} C_VEL
LIN {X 0,Y 411.233,Z 573.263,A -85,B 0,C 180,E1 -10680.643,E2 -10680.643} C_VEL
LIN {X 0,Y 411.238,Z 573.257,A -85,B 0,C 180,E1 -10683.618,E2 -10683.618} C_VEL
LIN {X 0,Y 411.203,Z 573.265,A -85,B 0,C 180,E1 -10686.852,E2 -10686.852} C_VEL
LIN {X 0,Y 411.215,Z 573.262,A -85,B 0,C 180,E1 -10690.05,E2 -10690.05} C_VEL
LIN {X 0,Y 411.263,Z 573.256,A -85,B 0,C 180,E1 -10693.13,E2 -10693.13} C_VEL
LIN {X 0,Y 411.313,Z 573.252,A -85,B 0,C 180,E1 -10696.89,E2 -10696.89} C_VEL
LIN {X 0,Y 411.307,Z 573.252,A -85,B 0,C 180,E1 -10700.161,E2 -10700.161} C_VEL
LIN {X 0,Y 411.46,Z 573.231,A -85,B 0,C 180,E1 -10703.132,E2 -10703.132} C_VEL
LIN {X 0,Y 411.312,Z 573.25,A -85,B 0,C 180,E1 -10705.098,E2 -10705.098} C_VEL
LIN {X 0,Y 411.483,Z 573.232,A -85,B 0,C 180,E1 -10707.613,E2 -10707.613} C_VEL
LIN {X 0,Y 415.081,Z 585.899,A -85,B 0,C 180,E1 -10708.516,E2 -10708.516} C_VEL
LIN {X 0,Y 415.406,Z 588.916,A -85,B 0,C 180,E1 -10708.745,E2 -10708.745} C_VEL
LIN {X 0,Y 414.895,Z 600.516,A -85,B 0,C 180,E1 -10709.686,E2 -10709.686} C_VEL
LIN {X 0,Y 414.246,Z 611.716,A -85,B 0,C 180,E1 -10710.85,E2 -10710.85} C_VEL
LIN {X 0,Y 413.622,Z 622.009,A -85,B 0,C 180,E1 -10712.19,E2 -10712.19} C_VEL
LIN {X 0,Y 412.94,Z 630.955,A -85,B 0,C 180,E1 -10713.658,E2 -10713.658} C_VEL
LIN {X 0,Y 412.474,Z 638.151,A -85,B 0,C 180,E1 -10715.131,E2 -10715.131} C_VEL
LIN {X 0,Y 412.127,Z 643.039,A -85,B 0,C 180,E1 -10716.363,E2 -10716.363} C_VEL
LIN {X 0,Y 411.721,Z 648.501,A -85,B 0,C 180,E1 -10718.093,E2 -10718.093} C_VEL
LIN {X 0,Y 411.377,Z 652.466,A -85,B 0,C 180,E1 -10719.836,E2 -10719.836} C_VEL
LIN {X 0,Y 411.258,Z 654.12,A -85,B 0,C 180,E1 -10720.834,E2 -10720.834} C_VEL
LIN {X 0,Y 411.185,Z 655.374,A -85,B 0,C 180,E1 -10721.835,E2 -10721.835} C_VEL
LIN {X 0,Y 411.181,Z 656.23,A -85,B 0,C 180,E1 -10722.91,E2 -10722.91} C_VEL
LIN {X 0,Y 410.557,Z 656.671,A -85,B 0,C 180,E1 -10723.727,E2 -10723.727} C_VEL
LIN {X 0,Y 407.749,Z 657.162,A -85,B 0,C 180,E1 -10725.058,E2 -10725.058} C_VEL
LIN {X 0,Y 404.96,Z 656.92,A -85,B 0,C 180,E1 -10726.401,E2 -10726.401} C_VEL
LIN {X 0,Y 404.378,Z 656.164,A -85,B 0,C 180,E1 -10727.227,E2 -10727.227} C_VEL
LIN {X 0,Y 404.559,Z 654.907,A -85,B 0,C 180,E1 -10728.221,E2 -10728.221} C_VEL
LIN {X 0,Y 404.91,Z 652.065,A -85,B 0,C 180,E1 -10729.782,E2 -10729.782} C_VEL
LIN {X 0,Y 405.365,Z 648.118,A -85,B 0,C 180,E1 -10731.35,E2 -10731.35} C_VEL
LIN {X 0,Y 406.046,Z 641.881,A -85,B 0,C 180,E1 -10733.188,E2 -10733.188} C_VEL
LIN {X 0,Y 406.768,Z 634.959,A -85,B 0,C 180,E1 -10734.769,E2 -10734.769} C_VEL
LIN {X 0,Y 407.552,Z 626.674,A -85,B 0,C 180,E1 -10736.272,E2 -10736.272} C_VEL
LIN {X 0,Y 408.446,Z 616.913,A -85,B 0,C 180,E1 -10737.682,E2 -10737.682} C_VEL
LIN {X 0,Y 409.167,Z 607.011,A -85,B 0,C 180,E1 -10738.838,E2 -10738.838} C_VEL
LIN {X 0,Y 409.924,Z 596.491,A -85,B 0,C 180,E1 -10739.813,E2 -10739.813} C_VEL
LIN {X 0,Y 410.039,Z 592.026,A -85,B 0,C 180,E1 -10740.177,E2 -10740.177} C_VEL
LIN {X 0,Y 406.541,Z 580.937,A -85,B 0,C 180,E1 -10741.153,E2 -10741.153} C_VEL
LIN {X 0,Y 404.124,Z 574.141,A -85,B 0,C 180,E1 -10741.692,E2 -10741.692} C_VEL
LIN {X 0,Y 404.179,Z 574.142,A -85,B 0,C 180,E1 -10745.015,E2 -10745.015} C_VEL
LIN {X 0,Y 404.227,Z 574.255,A -85,B 0,C 180,E1 -10748.029,E2 -10748.029} C_VEL
LIN {X 0,Y 405.11,Z 579.552,A -85,B 0,C 180,E1 -10750.242,E2 -10750.242} C_VEL
LIN {X 0,Y 405.402,Z 583.27,A -85,B 0,C 180,E1 -10751.803,E2 -10751.803} C_VEL
LIN {X 0,Y 405.197,Z 591.913,A -85,B 0,C 180,E1 -10755.325,E2 -10755.325} C_VEL
LIN {X 0,Y 404.96,Z 599.184,A -85,B 0,C 180,E1 -10758.265,E2 -10758.265} C_VEL
LIN {X 0,Y 404.703,Z 608.334,A -85,B 0,C 180,E1 -10761.978,E2 -10761.978} C_VEL
LIN {X 0,Y 404.47,Z 617.342,A -85,B 0,C 180,E1 -10765.618,E2 -10765.618} C_VEL
LIN {X 0,Y 404.154,Z 626.88,A -85,B 0,C 180,E1 -10769.44,E2 -10769.44} C_VEL
LIN {X 0,Y 407.442,Z 642.869,A -85,B 0,C 180,E1 -10770.141,E2 -10770.141} C_VEL
LIN {X 0,Y 408.234,Z 648.658,A -85,B 0,C 180,E1 -10770.447,E2 -10770.447} C_VEL
LIN {X 0,Y 407.584,Z 661.705,A -85,B 0,C 180,E1 -10771.214,E2 -10771.214} C_VEL
LIN {X 0,Y 406.991,Z 672.542,A -85,B 0,C 180,E1 -10772.04,E2 -10772.04} C_VEL
LIN {X 0,Y 406.185,Z 683.914,A -85,B 0,C 180,E1 -10773.127,E2 -10773.127} C_VEL
LIN {X 0,Y 405.524,Z 693.956,A -85,B 0,C 180,E1 -10774.325,E2 -10774.325} C_VEL
LIN {X 0,Y 404.836,Z 703.061,A -85,B 0,C 180,E1 -10775.651,E2 -10775.651} C_VEL
LIN {X 0,Y 404.184,Z 711.359,A -85,B 0,C 180,E1 -10777.153,E2 -10777.153} C_VEL
LIN {X 0,Y 403.744,Z 718.721,A -85,B 0,C 180,E1 -10778.827,E2 -10778.827} C_VEL
LIN {X 0,Y 403.423,Z 723.411,A -85,B 0,C 180,E1 -10780.17,E2 -10780.17} C_VEL
LIN {X 0,Y 403.174,Z 727.661,A -85,B 0,C 180,E1 -10781.714,E2 -10781.714} C_VEL
LIN {X 0,Y 402.969,Z 731.279,A -85,B 0,C 180,E1 -10783.578,E2 -10783.578} C_VEL
LIN {X 0,Y 402.878,Z 732.906,A -85,B 0,C 180,E1 -10784.831,E2 -10784.831} C_VEL
LIN {X 0,Y 402.838,Z 733.713,A -85,B 0,C 180,E1 -10785.863,E2 -10785.863} C_VEL
LIN {X 0,Y 402.931,Z 734.119,A -85,B 0,C 180,E1 -10787.617,E2 -10787.617} C_VEL
LIN {X 0,Y 402.959,Z 733.609,A -85,B 0,C 180,E1 -10788.94,E2 -10788.94} C_VEL
LIN {X 0,Y 402.969,Z 732.722,A -85,B 0,C 180,E1 -10789.956,E2 -10789.956} C_VEL
LIN {X 0,Y 403.09,Z 731.425,A -85,B 0,C 180,E1 -10790.972,E2 -10790.972} C_VEL
LIN {X 0,Y 403.337,Z 728.637,A -85,B 0,C 180,E1 -10792.491,E2 -10792.491} C_VEL
LIN {X 0,Y 403.565,Z 724.832,A -85,B 0,C 180,E1 -10794.003,E2 -10794.003} C_VEL
LIN {X 0,Y 403.925,Z 719.882,A -85,B 0,C 180,E1 -10795.51,E2 -10795.51} C_VEL
LIN {X 0,Y 404.423,Z 713.629,A -85,B 0,C 180,E1 -10797.012,E2 -10797.012} C_VEL
LIN {X 0,Y 405.129,Z 705.864,A -85,B 0,C 180,E1 -10798.509,E2 -10798.509} C_VEL
LIN {X 0,Y 405.834,Z 697.976,A -85,B 0,C 180,E1 -10799.752,E2 -10799.752} C_VEL
LIN {X 0,Y 406.66,Z 688.387,A -85,B 0,C 180,E1 -10800.991,E2 -10800.991} C_VEL
LIN {X 0,Y 407.625,Z 676.436,A -85,B 0,C 180,E1 -10802.224,E2 -10802.224} C_VEL
LIN {X 0,Y 408.45,Z 664.283,A -85,B 0,C 180,E1 -10803.206,E2 -10803.206} C_VEL
LIN {X 0,Y 409.261,Z 651.193,A -85,B 0,C 180,E1 -10804.011,E2 -10804.011} C_VEL
LIN {X 0,Y 409.015,Z 647.196,A -85,B 0,C 180,E1 -10804.233,E2 -10804.233} C_VEL
LIN {X 0,Y 406.032,Z 634.117,A -85,B 0,C 180,E1 -10804.948,E2 -10804.948} C_VEL
LIN {X 0,Y 404.624,Z 629.202,A -85,B 0,C 180,E1 -10805.201,E2 -10805.201} C_VEL
LIN {X 0,Y 404.969,Z 621.133,A -85,B 0,C 180,E1 -10808.437,E2 -10808.437} C_VEL
LIN {X 0,Y 405.169,Z 613.456,A -85,B 0,C 180,E1 -10811.507,E2 -10811.507} C_VEL
LIN {X 0,Y 405.477,Z 605.757,A -85,B 0,C 180,E1 -10814.556,E2 -10814.556} C_VEL
LIN {X 0,Y 405.789,Z 597.702,A -85,B 0,C 180,E1 -10817.723,E2 -10817.723} C_VEL
LIN {X 0,Y 406.005,Z 588.13,A -85,B 0,C 180,E1 -10821.316,E2 -10821.316} C_VEL
LIN {X 0,Y 405.896,Z 582.507,A -85,B 0,C 180,E1 -10823.469,E2 -10823.469} C_VEL
LIN {X 0,Y 404.489,Z 575.481,A -85,B 0,C 180,E1 -10826.3,E2 -10826.3} C_VEL
LIN {X 0,Y 404.189,Z 574.142,A -85,B 0,C 180,E1 -10826.878,E2 -10826.878} C_VEL
LIN {X 0,Y 404.148,Z 574.145,A -85,B 0,C 180,E1 -10830.285,E2 -10830.285} C_VEL
LIN {X 0,Y 404.139,Z 574.145,A -85,B 0,C 180,E1 -10833.813,E2 -10833.813} C_VEL
LIN {X 0,Y 404.136,Z 574.144,A -85,B 0,C 180,E1 -10836.877,E2 -10836.877} C_VEL
LIN {X 0,Y 404.163,Z 574.141,A -85,B 0,C 180,E1 -10840.085,E2 -10840.085} C_VEL
LIN {X 0,Y 404.201,Z 574.136,A -85,B 0,C 180,E1 -10843.093,E2 -10843.093} C_VEL
LIN {X 0,Y 404.219,Z 574.239,A -85,B 0,C 180,E1 -10845.61,E2 -10845.61} C_VEL
LIN {X 0,Y 405.993,Z 582.877,A -85,B 0,C 180,E1 -10848.869,E2 -10848.869} C_VEL
LIN {X 0,Y 407.541,Z 590.654,A -85,B 0,C 180,E1 -10851.626,E2 -10851.626} C_VEL
LIN {X 0,Y 408.023,Z 594.555,A -85,B 0,C 180,E1 -10852.927,E2 -10852.927} C_VEL
LIN {X 0,Y 407.398,Z 602.271,A -85,B 0,C 180,E1 -10855.301,E2 -10855.301} C_VEL
LIN {X 0,Y 406.362,Z 613.911,A -85,B 0,C 180,E1 -10858.746,E2 -10858.746} C_VEL
LIN {X 0,Y 405.557,Z 625.631,A -85,B 0,C 180,E1 -10862.104,E2 -10862.104} C_VEL
LIN {X 0,Y 404.837,Z 637.374,A -85,B 0,C 180,E1 -10865.378,E2 -10865.378} C_VEL
LIN {X 0,Y 404.28,Z 649.145,A -85,B 0,C 180,E1 -10868.59,E2 -10868.59} C_VEL
LIN {X 0,Y 403.862,Z 661.155,A -85,B 0,C 180,E1 -10871.791,E2 -10871.791} C_VEL
LIN {X 0,Y 405.732,Z 674.916,A -85,B 0,C 180,E1 -10872.271,E2 -10872.271} C_VEL
LIN {X 0,Y 406.818,Z 689.57,A -85,B 0,C 180,E1 -10872.922,E2 -10872.922} C_VEL
LIN {X 0,Y 407.489,Z 703.356,A -85,B 0,C 180,E1 -10873.725,E2 -10873.725} C_VEL
LIN {X 0,Y 406.672,Z 715.514,A -85,B 0,C 180,E1 -10874.592,E2 -10874.592} C_VEL
LIN {X 0,Y 405.847,Z 726.571,A -85,B 0,C 180,E1 -10875.587,E2 -10875.587} C_VEL
LIN {X 0,Y 405.074,Z 737.194,A -85,B 0,C 180,E1 -10876.779,E2 -10876.779} C_VEL
LIN {X 0,Y 404.367,Z 747.494,A -85,B 0,C 180,E1 -10878.217,E2 -10878.217} C_VEL
LIN {X 0,Y 403.744,Z 756.148,A -85,B 0,C 180,E1 -10879.723,E2 -10879.723} C_VEL
LIN {X 0,Y 403.387,Z 764.175,A -85,B 0,C 180,E1 -10881.485,E2 -10881.485} C_VEL
LIN {X 0,Y 403.185,Z 769.571,A -85,B 0,C 180,E1 -10882.992,E2 -10882.992} C_VEL
LIN {X 0,Y 403.075,Z 773.749,A -85,B 0,C 180,E1 -10884.498,E2 -10884.498} C_VEL
LIN {X 0,Y 403.008,Z 776.837,A -85,B 0,C 180,E1 -10886.001,E2 -10886.001} C_VEL
LIN {X 0,Y 403.069,Z 778.312,A -85,B 0,C 180,E1 -10887.003,E2 -10887.003} C_VEL
LIN {X 0,Y 403.084,Z 779.37,A -85,B 0,C 180,E1 -10888.003,E2 -10888.003} C_VEL
LIN {X 0,Y 403.086,Z 780.021,A -85,B 0,C 180,E1 -10889.002,E2 -10889.002} C_VEL
LIN {X 0,Y 403.12,Z 780.215,A -85,B 0,C 180,E1 -10890.001,E2 -10890.001} C_VEL
LIN {X 0,Y 403.1,Z 779.978,A -85,B 0,C 180,E1 -10891,E2 -10891} C_VEL
LIN {X 0,Y 403.084,Z 779.336,A -85,B 0,C 180,E1 -10891.999,E2 -10891.999} C_VEL
LIN {X 0,Y 403.081,Z 778.271,A -85,B 0,C 180,E1 -10892.999,E2 -10892.999} C_VEL
LIN {X 0,Y 402.998,Z 776.722,A -85,B 0,C 180,E1 -10894.001,E2 -10894.001} C_VEL
LIN {X 0,Y 403.098,Z 773.58,A -85,B 0,C 180,E1 -10895.504,E2 -10895.504} C_VEL
LIN {X 0,Y 403.115,Z 769.309,A -85,B 0,C 180,E1 -10897.011,E2 -10897.011} C_VEL
LIN {X 0,Y 403.408,Z 762.792,A -85,B 0,C 180,E1 -10898.769,E2 -10898.769} C_VEL
LIN {X 0,Y 403.73,Z 755.578,A -85,B 0,C 180,E1 -10900.279,E2 -10900.279} C_VEL
LIN {X 0,Y 404.318,Z 746.592,A -85,B 0,C 180,E1 -10901.786,E2 -10901.786} C_VEL
LIN {X 0,Y 404.976,Z 737.337,A -85,B 0,C 180,E1 -10903.039,E2 -10903.039} C_VEL
LIN {X 0,Y 405.543,Z 727.042,A -85,B 0,C 180,E1 -10904.17,E2 -10904.17} C_VEL
LIN {X 0,Y 406.302,Z 715.714,A -85,B 0,C 180,E1 -10905.167,E2 -10905.167} C_VEL
LIN {X 0,Y 407.023,Z 703.913,A -85,B 0,C 180,E1 -10905.974,E2 -10905.974} C_VEL
LIN {X 0,Y 406.94,Z 698.776,A -85,B 0,C 180,E1 -10906.274,E2 -10906.274} C_VEL
LIN {X 0,Y 406.036,Z 687.086,A -85,B 0,C 180,E1 -10906.849,E2 -10906.849} C_VEL
LIN {X 0,Y 404.413,Z 668.293,A -85,B 0,C 180,E1 -10907.547,E2 -10907.547} C_VEL
LIN {X 0,Y 403.783,Z 662.186,A -85,B 0,C 180,E1 -10907.718,E2 -10907.718} C_VEL
LIN {X 0,Y 404.2,Z 649.218,A -85,B 0,C 180,E1 -10911.149,E2 -10911.149} C_VEL
LIN {X 0,Y 404.731,Z 636.234,A -85,B 0,C 180,E1 -10914.63,E2 -10914.63} C_VEL
LIN {X 0,Y 405.417,Z 623.11,A -85,B 0,C 180,E1 -10918.19,E2 -10918.19} C_VEL
LIN {X 0,Y 406.116,Z 611.984,A -85,B 0,C 180,E1 -10921.277,E2 -10921.277} C_VEL
LIN {X 0,Y 406.965,Z 599.766,A -85,B 0,C 180,E1 -10924.743,E2 -10924.743} C_VEL
LIN {X 0,Y 407.396,Z 591.56,A -85,B 0,C 180,E1 -10927.142,E2 -10927.142} C_VEL
LIN {X 0,Y 406.229,Z 584.673,A -85,B 0,C 180,E1 -10929.31,E2 -10929.31} C_VEL
LIN {X 0,Y 404.5,Z 575.759,A -85,B 0,C 180,E1 -10932.251,E2 -10932.251} C_VEL
LIN {X 0,Y 404.151,Z 574.144,A -85,B 0,C 180,E1 -10932.847,E2 -10932.847} C_VEL
LIN {X 0,Y 404.153,Z 574.144,A -85,B 0,C 180,E1 -10935.926,E2 -10935.926} C_VEL
LIN {X 0,Y 404.124,Z 574.148,A -85,B 0,C 180,E1 -10938.635,E2 -10938.635} C_VEL
LIN {X 0,Y 404.163,Z 574.139,A -85,B 0,C 180,E1 -10941.491,E2 -10941.491} C_VEL
LIN {X 0,Y 404.191,Z 574.136,A -85,B 0,C 180,E1 -10944.984,E2 -10944.984} C_VEL
LIN {X 0,Y 404.147,Z 574.144,A -85,B 0,C 180,E1 -10948.554,E2 -10948.554} C_VEL
LIN {X 0,Y 404.2,Z 574.137,A -85,B 0,C 180,E1 -10952,E2 -10952} C_VEL
LIN {X 0,Y 404.182,Z 574.137,A -85,B 0,C 180,E1 -10955.334,E2 -10955.334} C_VEL
LIN {X 0,Y 404.143,Z 574.146,A -85,B 0,C 180,E1 -10958.58,E2 -10958.58} C_VEL
LIN {X 0,Y 404.215,Z 574.134,A -85,B 0,C 180,E1 -10961.762,E2 -10961.762} C_VEL
LIN {X 0,Y 404.211,Z 574.134,A -85,B 0,C 180,E1 -10964.882,E2 -10964.882} C_VEL
LIN {X 0,Y 404.261,Z 574.129,A -85,B 0,C 180,E1 -10967.958,E2 -10967.958} C_VEL
LIN {X 0,Y 404.438,Z 574.108,A -85,B 0,C 180,E1 -10972.099,E2 -10972.099} C_VEL
LIN {X 0,Y 404.428,Z 574.109,A -85,B 0,C 180,E1 -10974.015,E2 -10974.015} C_VEL
LIN {X 0,Y 404.484,Z 574.102,A -85,B 0,C 180,E1 -10978.008,E2 -10978.008} C_VEL
LIN {X 0,Y 404.615,Z 574.085,A -85,B 0,C 180,E1 -10980,E2 -10980} C_VEL
LIN {X 0,Y 404.418,Z 574.109,A -85,B 0,C 180,E1 -10982.988,E2 -10982.988} C_VEL
LIN {X 0,Y 404.415,Z 574.109,A -85,B 0,C 180,E1 -10986.987,E2 -10986.987} C_VEL
LIN {X 0,Y 404.261,Z 574.13,A -85,B 0,C 180,E1 -10990.011,E2 -10990.011} C_VEL
LIN {X 0,Y 404.27,Z 574.125,A -85,B 0,C 180,E1 -10993.211,E2 -10993.211} C_VEL
LIN {X 0,Y 404.219,Z 574.134,A -85,B 0,C 180,E1 -10997.006,E2 -10997.006} C_VEL
LIN {X 0,Y 404.167,Z 574.143,A -85,B 0,C 180,E1 -11000.351,E2 -11000.351} C_VEL
LIN {X 0,Y 404.172,Z 574.138,A -85,B 0,C 180,E1 -11003.574,E2 -11003.574} C_VEL
LIN {X 0,Y 404.186,Z 574.137,A -85,B 0,C 180,E1 -11005.766,E2 -11005.766} C_VEL
LIN {X 0,Y 404.198,Z 574.136,A -85,B 0,C 180,E1 -11007.999,E2 -11007.999} C_VEL
LIN {X 0,Y 404.141,Z 574.142,A -85,B 0,C 180,E1 -11011.557,E2 -11011.557} C_VEL
LIN {X 0,Y 404.187,Z 574.137,A -85,B 0,C 180,E1 -11015.015,E2 -11015.015} C_VEL
LIN {X 0,Y 404.159,Z 574.143,A -85,B 0,C 180,E1 -11018.756,E2 -11018.756} C_VEL
LIN {X 0,Y 404.125,Z 574.143,A -85,B 0,C 180,E1 -11021.599,E2 -11021.599} C_VEL
LIN {X 0,Y 404.151,Z 574.145,A -85,B 0,C 180,E1 -11024.522,E2 -11024.522} C_VEL
LIN {X 0,Y 404.141,Z 574.142,A -85,B 0,C 180,E1 -11027.295,E2 -11027.295} C_VEL
LIN {X 0,Y 404.17,Z 574.139,A -85,B 0,C 180,E1 -11029.955,E2 -11029.955} C_VEL
LIN {X 0,Y 404.137,Z 574.143,A -85,B 0,C 180,E1 -11033.124,E2 -11033.124} C_VEL
LIN {X 0,Y 404.145,Z 574.144,A -85,B 0,C 180,E1 -11036.187,E2 -11036.187} C_VEL
LIN {X 0,Y 404.146,Z 574.142,A -85,B 0,C 180,E1 -11039.714,E2 -11039.714} C_VEL
LIN {X 0,Y 404.195,Z 574.136,A -85,B 0,C 180,E1 -11043.122,E2 -11043.122} C_VEL
LIN {X 0,Y 404.177,Z 574.138,A -85,B 0,C 180,E1 -11045.334,E2 -11045.334} C_VEL
LIN {X 0,Y 404.16,Z 574.144,A -85,B 0,C 180,E1 -11048.581,E2 -11048.581} C_VEL
LIN {X 0,Y 404.21,Z 574.133,A -85,B 0,C 180,E1 -11051.761,E2 -11051.761} C_VEL
LIN {X 0,Y 404.208,Z 574.136,A -85,B 0,C 180,E1 -11054.881,E2 -11054.881} C_VEL
LIN {X 0,Y 404.269,Z 574.126,A -85,B 0,C 180,E1 -11057.958,E2 -11057.958} C_VEL
LIN {X 0,Y 404.432,Z 574.108,A -85,B 0,C 180,E1 -11062.099,E2 -11062.099} C_VEL
LIN {X 0,Y 404.423,Z 574.107,A -85,B 0,C 180,E1 -11064.014,E2 -11064.014} C_VEL
LIN {X 0,Y 404.47,Z 574.296,A -85,B 0,C 180,E1 -11067.385,E2 -11067.385} C_VEL
LIN {X 0,Y 407.817,Z 586.122,A -85,B 0,C 180,E1 -11068.223,E2 -11068.223} C_VEL
LIN {X 0,Y 408.478,Z 588.425,A -85,B 0,C 180,E1 -11068.416,E2 -11068.416} C_VEL
LIN {X 0,Y 408.156,Z 598.934,A -85,B 0,C 180,E1 -11069.254,E2 -11069.254} C_VEL
LIN {X 0,Y 407.545,Z 609.781,A -85,B 0,C 180,E1 -11070.328,E2 -11070.328} C_VEL
LIN {X 0,Y 406.975,Z 619.163,A -85,B 0,C 180,E1 -11071.483,E2 -11071.483} C_VEL
LIN {X 0,Y 406.221,Z 628.895,A -85,B 0,C 180,E1 -11072.974,E2 -11072.974} C_VEL
LIN {X 0,Y 405.673,Z 636.712,A -85,B 0,C 180,E1 -11074.47,E2 -11074.47} C_VEL
LIN {X 0,Y 405.186,Z 642.973,A -85,B 0,C 180,E1 -11075.973,E2 -11075.973} C_VEL
LIN {X 0,Y 404.827,Z 647.952,A -85,B 0,C 180,E1 -11077.48,E2 -11077.48} C_VEL
LIN {X 0,Y 404.49,Z 651.833,A -85,B 0,C 180,E1 -11078.996,E2 -11078.996} C_VEL
LIN {X 0,Y 404.32,Z 653.836,A -85,B 0,C 180,E1 -11080.009,E2 -11080.009} C_VEL
LIN {X 0,Y 404.213,Z 655.426,A -85,B 0,C 180,E1 -11081.025,E2 -11081.025} C_VEL
LIN {X 0,Y 404.149,Z 657.193,A -85,B 0,C 180,E1 -11082.902,E2 -11082.902} C_VEL
LIN {X 0,Y 404.122,Z 657.66,A -85,B 0,C 180,E1 -11084.09,E2 -11084.09} C_VEL
LIN {X 0,Y 404.168,Z 657.616,A -85,B 0,C 180,E1 -11085.118,E2 -11085.118} C_VEL
LIN {X 0,Y 404.352,Z 656.339,A -85,B 0,C 180,E1 -11087.071,E2 -11087.071} C_VEL
LIN {X 0,Y 404.378,Z 656.164,A -85,B 0,C 180,E1 -11087.227,E2 -11087.227} C_VEL
LIN {X 0,Y 403.845,Z 655.272,A -85,B 0,C 180,E1 -11088.049,E2 -11088.049} C_VEL
LIN {X 0,Y 401.302,Z 653.51,A -85,B 0,C 180,E1 -11089.391,E2 -11089.391} C_VEL
LIN {X 0,Y 399.206,Z 651.666,A -85,B 0,C 180,E1 -11090.459,E2 -11090.459} C_VEL
LIN {X 0,Y 398.431,Z 649.839,A -85,B 0,C 180,E1 -11091.261,E2 -11091.261} C_VEL
LIN {X 0,Y 398.436,Z 649.105,A -85,B 0,C 180,E1 -11091.526,E2 -11091.526} C_VEL
LIN {X 0,Y 398.901,Z 645.08,A -85,B 0,C 180,E1 -11092.804,E2 -11092.804} C_VEL
LIN {X 0,Y 399.611,Z 638.762,A -85,B 0,C 180,E1 -11094.411,E2 -11094.411} C_VEL
LIN {X 0,Y 400.502,Z 630.675,A -85,B 0,C 180,E1 -11096.02,E2 -11096.02} C_VEL
LIN {X 0,Y 401.33,Z 622.288,A -85,B 0,C 180,E1 -11097.365,E2 -11097.365} C_VEL
LIN {X 0,Y 402.155,Z 612.243,A -85,B 0,C 180,E1 -11098.675,E2 -11098.675} C_VEL
LIN {X 0,Y 403.029,Z 601.275,A -85,B 0,C 180,E1 -11099.799,E2 -11099.799} C_VEL
LIN {X 0,Y 403.434,Z 594.945,A -85,B 0,C 180,E1 -11100.343,E2 -11100.343} C_VEL
LIN {X 0,Y 401.67,Z 588.147,A -85,B 0,C 180,E1 -11100.981,E2 -11100.981} C_VEL
LIN {X 0,Y 398.112,Z 578.196,A -85,B 0,C 180,E1 -11101.836,E2 -11101.836} C_VEL
LIN {X 0,Y 397.089,Z 575.02,A -85,B 0,C 180,E1 -11102.088,E2 -11102.088} C_VEL
LIN {X 0,Y 397.114,Z 575.02,A -85,B 0,C 180,E1 -11105.503,E2 -11105.503} C_VEL
LIN {X 0,Y 397.159,Z 575.196,A -85,B 0,C 180,E1 -11107.834,E2 -11107.834} C_VEL
LIN {X 0,Y 398.107,Z 580.51,A -85,B 0,C 180,E1 -11110.057,E2 -11110.057} C_VEL
LIN {X 0,Y 398.377,Z 585.543,A -85,B 0,C 180,E1 -11112.189,E2 -11112.189} C_VEL
LIN {X 0,Y 398.169,Z 594.28,A -85,B 0,C 180,E1 -11115.778,E2 -11115.778} C_VEL
LIN {X 0,Y 397.913,Z 601.01,A -85,B 0,C 180,E1 -11118.53,E2 -11118.53} C_VEL
LIN {X 0,Y 397.659,Z 610.245,A -85,B 0,C 180,E1 -11122.288,E2 -11122.288} C_VEL
LIN {X 0,Y 397.399,Z 619.884,A -85,B 0,C 180,E1 -11126.219,E2 -11126.219} C_VEL
LIN {X 0,Y 397.143,Z 627.371,A -85,B 0,C 180,E1 -11129.19,E2 -11129.19} C_VEL
LIN {X 0,Y 399.886,Z 640.547,A -85,B 0,C 180,E1 -11129.748,E2 -11129.748} C_VEL
LIN {X 0,Y 401.379,Z 649.032,A -85,B 0,C 180,E1 -11130.204,E2 -11130.204} C_VEL
LIN {X 0,Y 400.737,Z 661.253,A -85,B 0,C 180,E1 -11130.929,E2 -11130.929} C_VEL
LIN {X 0,Y 400.077,Z 672.958,A -85,B 0,C 180,E1 -11131.83,E2 -11131.83} C_VEL
LIN {X 0,Y 399.247,Z 684.056,A -85,B 0,C 180,E1 -11132.905,E2 -11132.905} C_VEL
LIN {X 0,Y 398.519,Z 694.492,A -85,B 0,C 180,E1 -11134.171,E2 -11134.171} C_VEL
LIN {X 0,Y 397.842,Z 703.283,A -85,B 0,C 180,E1 -11135.473,E2 -11135.473} C_VEL
LIN {X 0,Y 397.137,Z 712.044,A -85,B 0,C 180,E1 -11137.088,E2 -11137.088} C_VEL
LIN {X 0,Y 396.708,Z 719.023,A -85,B 0,C 180,E1 -11138.705,E2 -11138.705} C_VEL
LIN {X 0,Y 396.323,Z 724.476,A -85,B 0,C 180,E1 -11140.311,E2 -11140.311} C_VEL
LIN {X 0,Y 396.083,Z 728.613,A -85,B 0,C 180,E1 -11141.91,E2 -11141.91} C_VEL
LIN {X 0,Y 395.895,Z 731.6,A -85,B 0,C 180,E1 -11143.499,E2 -11143.499} C_VEL
LIN {X 0,Y 395.815,Z 732.998,A -85,B 0,C 180,E1 -11144.554,E2 -11144.554} C_VEL
LIN {X 0,Y 395.761,Z 733.972,A -85,B 0,C 180,E1 -11145.605,E2 -11145.605} C_VEL
LIN {X 0,Y 395.848,Z 734.553,A -85,B 0,C 180,E1 -11147.544,E2 -11147.544} C_VEL
LIN {X 0,Y 395.892,Z 734.212,A -85,B 0,C 180,E1 -11148.74,E2 -11148.74} C_VEL
LIN {X 0,Y 395.88,Z 733.441,A -85,B 0,C 180,E1 -11149.775,E2 -11149.775} C_VEL
LIN {X 0,Y 396.012,Z 732.236,A -85,B 0,C 180,E1 -11150.81,E2 -11150.81} C_VEL
LIN {X 0,Y 396.256,Z 729.631,A -85,B 0,C 180,E1 -11152.356,E2 -11152.356} C_VEL
LIN {X 0,Y 396.497,Z 726.014,A -85,B 0,C 180,E1 -11153.895,E2 -11153.895} C_VEL
LIN {X 0,Y 396.857,Z 721.278,A -85,B 0,C 180,E1 -11155.43,E2 -11155.43} C_VEL
LIN {X 0,Y 397.406,Z 715.289,A -85,B 0,C 180,E1 -11156.959,E2 -11156.959} C_VEL
LIN {X 0,Y 398.095,Z 707.812,A -85,B 0,C 180,E1 -11158.483,E2 -11158.483} C_VEL
LIN {X 0,Y 398.982,Z 698.562,A -85,B 0,C 180,E1 -11160,E2 -11160} C_VEL
LIN {X 0,Y 399.874,Z 689.055,A -85,B 0,C 180,E1 -11161.259,E2 -11161.259} C_VEL
LIN {X 0,Y 400.814,Z 678.109,A -85,B 0,C 180,E1 -11162.425,E2 -11162.425} C_VEL
LIN {X 0,Y 401.623,Z 666.982,A -85,B 0,C 180,E1 -11163.379,E2 -11163.379} C_VEL
LIN {X 0,Y 402.403,Z 655.884,A -85,B 0,C 180,E1 -11164.119,E2 -11164.119} C_VEL
LIN {X 0,Y 402.647,Z 650.169,A -85,B 0,C 180,E1 -11164.438,E2 -11164.438} C_VEL
LIN {X 0,Y 399.631,Z 636.32,A -85,B 0,C 180,E1 -11165.255,E2 -11165.255} C_VEL
LIN {X 0,Y 397.798,Z 629.693,A -85,B 0,C 180,E1 -11165.608,E2 -11165.608} C_VEL
LIN {X 0,Y 398.105,Z 620.97,A -85,B 0,C 180,E1 -11169.142,E2 -11169.142} C_VEL
LIN {X 0,Y 398.382,Z 612.033,A -85,B 0,C 180,E1 -11172.74,E2 -11172.74} C_VEL
LIN {X 0,Y 398.712,Z 604.237,A -85,B 0,C 180,E1 -11175.856,E2 -11175.856} C_VEL
LIN {X 0,Y 399,Z 596.31,A -85,B 0,C 180,E1 -11179.018,E2 -11179.018} C_VEL
LIN {X 0,Y 399.257,Z 587.869,A -85,B 0,C 180,E1 -11182.239,E2 -11182.239} C_VEL
LIN {X 0,Y 398.969,Z 583.665,A -85,B 0,C 180,E1 -11183.901,E2 -11183.901} C_VEL
LIN {X 0,Y 397.535,Z 576.73,A -85,B 0,C 180,E1 -11186.796,E2 -11186.796} C_VEL
LIN {X 0,Y 397.192,Z 575.012,A -85,B 0,C 180,E1 -11187.534,E2 -11187.534} C_VEL
LIN {X 0,Y 397.079,Z 575.027,A -85,B 0,C 180,E1 -11190.883,E2 -11190.883} C_VEL
LIN {X 0,Y 397.121,Z 575.021,A -85,B 0,C 180,E1 -11194.494,E2 -11194.494} C_VEL
LIN {X 0,Y 397.105,Z 575.02,A -85,B 0,C 180,E1 -11198.275,E2 -11198.275} C_VEL
LIN {X 0,Y 397.152,Z 575.009,A -85,B 0,C 180,E1 -11201.995,E2 -11201.995} C_VEL
LIN {X 0,Y 397.168,Z 575.155,A -85,B 0,C 180,E1 -11205.147,E2 -11205.147} C_VEL
LIN {X 0,Y 398.931,Z 583.714,A -85,B 0,C 180,E1 -11208.483,E2 -11208.483} C_VEL
LIN {X 0,Y 400.253,Z 590.056,A -85,B 0,C 180,E1 -11210.795,E2 -11210.795} C_VEL
LIN {X 0,Y 401.085,Z 595.881,A -85,B 0,C 180,E1 -11212.807,E2 -11212.807} C_VEL
LIN {X 0,Y 400.466,Z 603.414,A -85,B 0,C 180,E1 -11215.178,E2 -11215.178} C_VEL
LIN {X 0,Y 399.367,Z 615.173,A -85,B 0,C 180,E1 -11218.727,E2 -11218.727} C_VEL
LIN {X 0,Y 398.482,Z 627.327,A -85,B 0,C 180,E1 -11222.274,E2 -11222.274} C_VEL
LIN {X 0,Y 397.666,Z 640.497,A -85,B 0,C 180,E1 -11226.017,E2 -11226.017} C_VEL
LIN {X 0,Y 396.988,Z 655.012,A -85,B 0,C 180,E1 -11230.046,E2 -11230.046} C_VEL
LIN {X 0,Y 396.828,Z 659.88,A -85,B 0,C 180,E1 -11231.378,E2 -11231.378} C_VEL
LIN {X 0,Y 399.234,Z 677.883,A -85,B 0,C 180,E1 -11232.043,E2 -11232.043} C_VEL
LIN {X 0,Y 400.134,Z 691.801,A -85,B 0,C 180,E1 -11232.694,E2 -11232.694} C_VEL
LIN {X 0,Y 400.694,Z 703.766,A -85,B 0,C 180,E1 -11233.441,E2 -11233.441} C_VEL
LIN {X 0,Y 399.823,Z 715.665,A -85,B 0,C 180,E1 -11234.321,E2 -11234.321} C_VEL
LIN {X 0,Y 398.962,Z 726.545,A -85,B 0,C 180,E1 -11235.333,E2 -11235.333} C_VEL
LIN {X 0,Y 398.116,Z 737.21,A -85,B 0,C 180,E1 -11236.566,E2 -11236.566} C_VEL
LIN {X 0,Y 397.376,Z 747.301,A -85,B 0,C 180,E1 -11238.007,E2 -11238.007} C_VEL
LIN {X 0,Y 396.716,Z 755.898,A -85,B 0,C 180,E1 -11239.539,E2 -11239.539} C_VEL
LIN {X 0,Y 396.378,Z 762.848,A -85,B 0,C 180,E1 -11241.076,E2 -11241.076} C_VEL
LIN {X 0,Y 396.098,Z 769.24,A -85,B 0,C 180,E1 -11242.866,E2 -11242.866} C_VEL
LIN {X 0,Y 395.973,Z 773.386,A -85,B 0,C 180,E1 -11244.399,E2 -11244.399} C_VEL
LIN {X 0,Y 395.926,Z 776.459,A -85,B 0,C 180,E1 -11245.929,E2 -11245.929} C_VEL
LIN {X 0,Y 395.968,Z 777.926,A -85,B 0,C 180,E1 -11246.949,E2 -11246.949} C_VEL
LIN {X 0,Y 396.009,Z 778.98,A -85,B 0,C 180,E1 -11247.967,E2 -11247.967} C_VEL
LIN {X 0,Y 396.003,Z 779.619,A -85,B 0,C 180,E1 -11248.984,E2 -11248.984} C_VEL
LIN {X 0,Y 396.034,Z 779.794,A -85,B 0,C 180,E1 -11250.001,E2 -11250.001} C_VEL
LIN {X 0,Y 396.016,Z 779.548,A -85,B 0,C 180,E1 -11251.018,E2 -11251.018} C_VEL
LIN {X 0,Y 396.01,Z 778.896,A -85,B 0,C 180,E1 -11252.035,E2 -11252.035} C_VEL
LIN {X 0,Y 395.981,Z 777.804,A -85,B 0,C 180,E1 -11253.053,E2 -11253.053} C_VEL
LIN {X 0,Y 395.917,Z 776.24,A -85,B 0,C 180,E1 -11254.073,E2 -11254.073} C_VEL
LIN {X 0,Y 395.993,Z 773.066,A -85,B 0,C 180,E1 -11255.603,E2 -11255.603} C_VEL
LIN {X 0,Y 396.06,Z 768.764,A -85,B 0,C 180,E1 -11257.136,E2 -11257.136} C_VEL
LIN {X 0,Y 396.318,Z 763.23,A -85,B 0,C 180,E1 -11258.67,E2 -11258.67} C_VEL
LIN {X 0,Y 396.617,Z 756.276,A -85,B 0,C 180,E1 -11260.207,E2 -11260.207} C_VEL
LIN {X 0,Y 397.187,Z 747.523,A -85,B 0,C 180,E1 -11261.742,E2 -11261.742} C_VEL
LIN {X 0,Y 397.941,Z 737.587,A -85,B 0,C 180,E1 -11263.144,E2 -11263.144} C_VEL
LIN {X 0,Y 398.533,Z 727.453,A -85,B 0,C 180,E1 -11264.294,E2 -11264.294} C_VEL
LIN {X 0,Y 399.299,Z 716.306,A -85,B 0,C 180,E1 -11265.309,E2 -11265.309} C_VEL
LIN {X 0,Y 400.06,Z 704.881,A -85,B 0,C 180,E1 -11266.129,E2 -11266.129} C_VEL
LIN {X 0,Y 400.032,Z 699.899,A -85,B 0,C 180,E1 -11266.433,E2 -11266.433} C_VEL
LIN {X 0,Y 399.269,Z 689.136,A -85,B 0,C 180,E1 -11267.002,E2 -11267.002} C_VEL
LIN {X 0,Y 397.608,Z 669.633,A -85,B 0,C 180,E1 -11267.745,E2 -11267.745} C_VEL
LIN {X 0,Y 396.743,Z 661.235,A -85,B 0,C 180,E1 -11267.986,E2 -11267.986} C_VEL
LIN {X 0,Y 397.115,Z 649.089,A -85,B 0,C 180,E1 -11271.273,E2 -11271.273} C_VEL
LIN {X 0,Y 397.646,Z 637.104,A -85,B 0,C 180,E1 -11274.541,E2 -11274.541} C_VEL
LIN {X 0,Y 398.355,Z 624.291,A -85,B 0,C 180,E1 -11278.099,E2 -11278.099} C_VEL
LIN {X 0,Y 399.084,Z 612.932,A -85,B 0,C 180,E1 -11281.3,E2 -11281.3} C_VEL
LIN {X 0,Y 399.955,Z 600.746,A -85,B 0,C 180,E1 -11284.826,E2 -11284.826} C_VEL
LIN {X 0,Y 400.418,Z 592.777,A -85,B 0,C 180,E1 -11287.199,E2 -11287.199} C_VEL
LIN {X 0,Y 398.884,Z 584.099,A -85,B 0,C 180,E1 -11289.999,E2 -11289.999} C_VEL
LIN {X 0,Y 397.142,Z 575.018,A -85,B 0,C 180,E1 -11293.102,E2 -11293.102} C_VEL
LIN {X 0,Y 397.107,Z 575.022,A -85,B 0,C 180,E1 -11296.521,E2 -11296.521} C_VEL
LIN {X 0,Y 397.12,Z 575.02,A -85,B 0,C 180,E1 -11300.423,E2 -11300.423} C_VEL
LIN {X 0,Y 397.114,Z 575.021,A -85,B 0,C 180,E1 -11304.266,E2 -11304.266} C_VEL
LIN {X 0,Y 397.119,Z 575.019,A -85,B 0,C 180,E1 -11306.727,E2 -11306.727} C_VEL
LIN {X 0,Y 397.129,Z 575.019,A -85,B 0,C 180,E1 -11310.296,E2 -11310.296} C_VEL
LIN {X 0,Y 397.199,Z 575.01,A -85,B 0,C 180,E1 -11312.61,E2 -11312.61} C_VEL
LIN {X 0,Y 397.138,Z 575.017,A -85,B 0,C 180,E1 -11315.982,E2 -11315.982} C_VEL
LIN {X 0,Y 397.143,Z 575.014,A -85,B 0,C 180,E1 -11319.704,E2 -11319.704} C_VEL
LIN {X 0,Y 397.187,Z 575.01,A -85,B 0,C 180,E1 -11322.845,E2 -11322.845} C_VEL
LIN {X 0,Y 397.233,Z 575.005,A -85,B 0,C 180,E1 -11326.702,E2 -11326.702} C_VEL
LIN {X 0,Y 397.222,Z 575.005,A -85,B 0,C 180,E1 -11329.809,E2 -11329.809} C_VEL
LIN {X 0,Y 397.369,Z 574.987,A -85,B 0,C 180,E1 -11332.888,E2 -11332.888} C_VEL
LIN {X 0,Y 397.258,Z 575.001,A -85,B 0,C 180,E1 -11334.925,E2 -11334.925} C_VEL
LIN {X 0,Y 397.453,Z 574.977,A -85,B 0,C 180,E1 -11337.973,E2 -11337.973} C_VEL
LIN {X 0,Y 397.585,Z 574.96,A -85,B 0,C 180,E1 -11340,E2 -11340} C_VEL
LIN {X 0,Y 397.378,Z 574.985,A -85,B 0,C 180,E1 -11343.041,E2 -11343.041} C_VEL
LIN {X 0,Y 397.368,Z 574.986,A -85,B 0,C 180,E1 -11347.111,E2 -11347.111} C_VEL
LIN {X 0,Y 397.221,Z 575.007,A -85,B 0,C 180,E1 -11350.191,E2 -11350.191} C_VEL
LIN {X 0,Y 397.23,Z 575.002,A -85,B 0,C 180,E1 -11353.32,E2 -11353.32} C_VEL
LIN {X 0,Y 397.185,Z 575.009,A -85,B 0,C 180,E1 -11357.155,E2 -11357.155} C_VEL
LIN {X 0,Y 397.105,Z 575.021,A -85,B 0,C 180,E1 -11360.729,E2 -11360.729} C_VEL
LIN {X 0,Y 397.136,Z 575.017,A -85,B 0,C 180,E1 -11364.018,E2 -11364.018} C_VEL
LIN {X 0,Y 397.197,Z 575.006,A -85,B 0,C 180,E1 -11367.389,E2 -11367.389} C_VEL
LIN {X 0,Y 397.081,Z 575.024,A -85,B 0,C 180,E1 -11370.882,E2 -11370.882} C_VEL
LIN {X 0,Y 397.128,Z 575.02,A -85,B 0,C 180,E1 -11374.493,E2 -11374.493} C_VEL
LIN {X 0,Y 397.107,Z 575.021,A -85,B 0,C 180,E1 -11378.274,E2 -11378.274} C_VEL
LIN {X 0,Y 397.09,Z 575.022,A -85,B 0,C 180,E1 -11380.908,E2 -11380.908} C_VEL
LIN {X 0,Y 397.105,Z 575.018,A -85,B 0,C 180,E1 -11383.647,E2 -11383.647} C_VEL
LIN {X 0,Y 397.106,Z 575.023,A -85,B 0,C 180,E1 -11386.52,E2 -11386.52} C_VEL
LIN {X 0,Y 397.115,Z 575.022,A -85,B 0,C 180,E1 -11390.422,E2 -11390.422} C_VEL
LIN {X 0,Y 397.108,Z 575.022,A -85,B 0,C 180,E1 -11394.265,E2 -11394.265} C_VEL
LIN {X 0,Y 397.115,Z 575.021,A -85,B 0,C 180,E1 -11396.726,E2 -11396.726} C_VEL
LIN {X 0,Y 397.125,Z 575.019,A -85,B 0,C 180,E1 -11400.295,E2 -11400.295} C_VEL
LIN {X 0,Y 397.194,Z 575.011,A -85,B 0,C 180,E1 -11402.609,E2 -11402.609} C_VEL
LIN {X 0,Y 397.133,Z 575.016,A -85,B 0,C 180,E1 -11405.981,E2 -11405.981} C_VEL
LIN {X 0,Y 397.138,Z 575.013,A -85,B 0,C 180,E1 -11409.704,E2 -11409.704} C_VEL
LIN {X 0,Y 397.181,Z 575.012,A -85,B 0,C 180,E1 -11412.844,E2 -11412.844} C_VEL
LIN {X 0,Y 397.226,Z 575.008,A -85,B 0,C 180,E1 -11416.678,E2 -11416.678} C_VEL
LIN {X 0,Y 397.228,Z 575.003,A -85,B 0,C 180,E1 -11419.808,E2 -11419.808} C_VEL
LIN {X 0,Y 397.363,Z 574.989,A -85,B 0,C 180,E1 -11422.887,E2 -11422.887} C_VEL
LIN {X 0,Y 397.256,Z 575.002,A -85,B 0,C 180,E1 -11424.924,E2 -11424.924} C_VEL
LIN {X 0,Y 397.387,Z 574.988,A -85,B 0,C 180,E1 -11427.116,E2 -11427.116} C_VEL
LIN {X 0,Y 400.84,Z 587.099,A -85,B 0,C 180,E1 -11427.99,E2 -11427.99} C_VEL
LIN {X 0,Y 401.676,Z 590.387,A -85,B 0,C 180,E1 -11428.266,E2 -11428.266} C_VEL
LIN {X 0,Y 401.167,Z 602.288,A -85,B 0,C 180,E1 -11429.258,E2 -11429.258} C_VEL
LIN {X 0,Y 400.598,Z 612.079,A -85,B 0,C 180,E1 -11430.287,E2 -11430.287} C_VEL
LIN {X 0,Y 399.964,Z 621.54,A -85,B 0,C 180,E1 -11431.509,E2 -11431.509} C_VEL
LIN {X 0,Y 399.287,Z 629.592,A -85,B 0,C 180,E1 -11432.773,E2 -11432.773} C_VEL
LIN {X 0,Y 398.724,Z 637.464,A -85,B 0,C 180,E1 -11434.295,E2 -11434.295} C_VEL
LIN {X 0,Y 398.283,Z 642.815,A -85,B 0,C 180,E1 -11435.568,E2 -11435.568} C_VEL
LIN {X 0,Y 397.902,Z 648.051,A -85,B 0,C 180,E1 -11437.101,E2 -11437.101} C_VEL
LIN {X 0,Y 397.558,Z 652.026,A -85,B 0,C 180,E1 -11438.59,E2 -11438.59} C_VEL
LIN {X 0,Y 397.273,Z 655.206,A -85,B 0,C 180,E1 -11440.189,E2 -11440.189} C_VEL
LIN {X 0,Y 397.181,Z 656.704,A -85,B 0,C 180,E1 -11441.223,E2 -11441.223} C_VEL
LIN {X 0,Y 397.137,Z 658.424,A -85,B 0,C 180,E1 -11443.299,E2 -11443.299} C_VEL
LIN {X 0,Y 397.112,Z 658.715,A -85,B 0,C 180,E1 -11444.344,E2 -11444.344} C_VEL
LIN {X 0,Y 397.153,Z 658.558,A -85,B 0,C 180,E1 -11445.392,E2 -11445.392} C_VEL
LIN {X 0,Y 397.384,Z 657.247,A -85,B 0,C 180,E1 -11447.276,E2 -11447.276} C_VEL
LIN {X 0,Y 397.629,Z 655.613,A -85,B 0,C 180,E1 -11448.55,E2 -11448.55} C_VEL
LIN {X 0,Y 398.02,Z 652.632,A -85,B 0,C 180,E1 -11450.139,E2 -11450.139} C_VEL
LIN {X 0,Y 398.436,Z 649.105,A -85,B 0,C 180,E1 -11451.526,E2 -11451.526} C_VEL
LIN {X 0,Y 398.066,Z 646.916,A -85,B 0,C 180,E1 -11452.315,E2 -11452.315} C_VEL
LIN {X 0,Y 395.791,Z 643.157,A -85,B 0,C 180,E1 -11453.6,E2 -11453.6} C_VEL
LIN {X 0,Y 393.565,Z 638.723,A -85,B 0,C 180,E1 -11454.847,E2 -11454.847} C_VEL
LIN {X 0,Y 393.264,Z 635.478,A -85,B 0,C 180,E1 -11455.565,E2 -11455.565} C_VEL
LIN {X 0,Y 394.274,Z 626.532,A -85,B 0,C 180,E1 -11457.159,E2 -11457.159} C_VEL
LIN {X 0,Y 395.105,Z 617.847,A -85,B 0,C 180,E1 -11458.411,E2 -11458.411} C_VEL
LIN {X 0,Y 396.012,Z 606.901,A -85,B 0,C 180,E1 -11459.676,E2 -11459.676} C_VEL
LIN {X 0,Y 396.78,Z 596.743,A -85,B 0,C 180,E1 -11460.612,E2 -11460.612} C_VEL
LIN {X 0,Y 394.871,Z 589.544,A -85,B 0,C 180,E1 -11461.317,E2 -11461.317} C_VEL
LIN {X 0,Y 390.8,Z 578.291,A -85,B 0,C 180,E1 -11462.304,E2 -11462.304} C_VEL
LIN {X 0,Y 390.065,Z 575.899,A -85,B 0,C 180,E1 -11462.505,E2 -11462.505} C_VEL
LIN {X 0,Y 390.052,Z 575.9,A -85,B 0,C 180,E1 -11465.825,E2 -11465.825} C_VEL
LIN {X 0,Y 390.105,Z 575.994,A -85,B 0,C 180,E1 -11467.563,E2 -11467.563} C_VEL
LIN {X 0,Y 391.204,Z 582.394,A -85,B 0,C 180,E1 -11470.295,E2 -11470.295} C_VEL
LIN {X 0,Y 391.385,Z 587.818,A -85,B 0,C 180,E1 -11472.59,E2 -11472.59} C_VEL
LIN {X 0,Y 391.173,Z 595.937,A -85,B 0,C 180,E1 -11475.942,E2 -11475.942} C_VEL
LIN {X 0,Y 390.843,Z 603.454,A -85,B 0,C 180,E1 -11479.043,E2 -11479.043} C_VEL
LIN {X 0,Y 390.647,Z 611.457,A -85,B 0,C 180,E1 -11482.332,E2 -11482.332} C_VEL
LIN {X 0,Y 390.394,Z 620.614,A -85,B 0,C 180,E1 -11486.078,E2 -11486.078} C_VEL
LIN {X 0,Y 390.106,Z 627.557,A -85,B 0,C 180,E1 -11488.911,E2 -11488.911} C_VEL
LIN {X 0,Y 393.02,Z 641.89,A -85,B 0,C 180,E1 -11489.54,E2 -11489.54} C_VEL
LIN {X 0,Y 394.494,Z 649.885,A -85,B 0,C 180,E1 -11489.986,E2 -11489.986} C_VEL
LIN {X 0,Y 393.818,Z 662.262,A -85,B 0,C 180,E1 -11490.744,E2 -11490.744} C_VEL
LIN {X 0,Y 393.059,Z 674.502,A -85,B 0,C 180,E1 -11491.717,E2 -11491.717} C_VEL
LIN {X 0,Y 392.237,Z 685.327,A -85,B 0,C 180,E1 -11492.813,E2 -11492.813} C_VEL
LIN {X 0,Y 391.479,Z 695.435,A -85,B 0,C 180,E1 -11494.075,E2 -11494.075} C_VEL
LIN {X 0,Y 390.84,Z 703.438,A -85,B 0,C 180,E1 -11495.287,E2 -11495.287} C_VEL
LIN {X 0,Y 390.19,Z 711.253,A -85,B 0,C 180,E1 -11496.718,E2 -11496.718} C_VEL
LIN {X 0,Y 389.74,Z 718.215,A -85,B 0,C 180,E1 -11498.305,E2 -11498.305} C_VEL
LIN {X 0,Y 389.326,Z 723.935,A -85,B 0,C 180,E1 -11499.942,E2 -11499.942} C_VEL
LIN {X 0,Y 389.056,Z 728.336,A -85,B 0,C 180,E1 -11501.572,E2 -11501.572} C_VEL
LIN {X 0,Y 388.832,Z 731.76,A -85,B 0,C 180,E1 -11503.322,E2 -11503.322} C_VEL
LIN {X 0,Y 388.675,Z 734.142,A -85,B 0,C 180,E1 -11505.337,E2 -11505.337} C_VEL
LIN {X 0,Y 388.7,Z 734.803,A -85,B 0,C 180,E1 -11506.406,E2 -11506.406} C_VEL
LIN {X 0,Y 388.76,Z 734.99,A -85,B 0,C 180,E1 -11507.471,E2 -11507.471} C_VEL
LIN {X 0,Y 388.794,Z 734.756,A -85,B 0,C 180,E1 -11508.531,E2 -11508.531} C_VEL
LIN {X 0,Y 388.794,Z 734.129,A -85,B 0,C 180,E1 -11509.586,E2 -11509.586} C_VEL
LIN {X 0,Y 388.904,Z 733.052,A -85,B 0,C 180,E1 -11510.64,E2 -11510.64} C_VEL
LIN {X 0,Y 389.083,Z 731.53,A -85,B 0,C 180,E1 -11511.692,E2 -11511.692} C_VEL
LIN {X 0,Y 389.334,Z 728.766,A -85,B 0,C 180,E1 -11513.12,E2 -11513.12} C_VEL
LIN {X 0,Y 389.662,Z 724.292,A -85,B 0,C 180,E1 -11514.826,E2 -11514.826} C_VEL
LIN {X 0,Y 390.146,Z 718.987,A -85,B 0,C 180,E1 -11516.386,E2 -11516.386} C_VEL
LIN {X 0,Y 390.792,Z 712.362,A -85,B 0,C 180,E1 -11517.939,E2 -11517.939} C_VEL
LIN {X 0,Y 391.667,Z 704.071,A -85,B 0,C 180,E1 -11519.486,E2 -11519.486} C_VEL
LIN {X 0,Y 392.506,Z 695.651,A -85,B 0,C 180,E1 -11520.77,E2 -11520.77} C_VEL
LIN {X 0,Y 393.498,Z 685.384,A -85,B 0,C 180,E1 -11522.047,E2 -11522.047} C_VEL
LIN {X 0,Y 394.517,Z 673.577,A -85,B 0,C 180,E1 -11523.212,E2 -11523.212} C_VEL
LIN {X 0,Y 395.353,Z 662.591,A -85,B 0,C 180,E1 -11524.078,E2 -11524.078} C_VEL
LIN {X 0,Y 396.013,Z 651.543,A -85,B 0,C 180,E1 -11524.762,E2 -11524.762} C_VEL
LIN {X 0,Y 393.101,Z 638.219,A -85,B 0,C 180,E1 -11525.595,E2 -11525.595} C_VEL
LIN {X 0,Y 390.842,Z 630.206,A -85,B 0,C 180,E1 -11526.032,E2 -11526.032} C_VEL
LIN {X 0,Y 391.204,Z 622.23,A -85,B 0,C 180,E1 -11529.305,E2 -11529.305} C_VEL
LIN {X 0,Y 391.515,Z 613.258,A -85,B 0,C 180,E1 -11532.967,E2 -11532.967} C_VEL
LIN {X 0,Y 391.89,Z 605.549,A -85,B 0,C 180,E1 -11536.14,E2 -11536.14} C_VEL
LIN {X 0,Y 392.183,Z 597.389,A -85,B 0,C 180,E1 -11539.362,E2 -11539.362} C_VEL
LIN {X 0,Y 392.44,Z 590.446,A -85,B 0,C 180,E1 -11542.091,E2 -11542.091} C_VEL
LIN {X 0,Y 392.229,Z 585.854,A -85,B 0,C 180,E1 -11543.964,E2 -11543.964} C_VEL
LIN {X 0,Y 390.962,Z 579.495,A -85,B 0,C 180,E1 -11546.706,E2 -11546.706} C_VEL
LIN {X 0,Y 390.09,Z 575.896,A -85,B 0,C 180,E1 -11548.356,E2 -11548.356} C_VEL
LIN {X 0,Y 390.028,Z 575.905,A -85,B 0,C 180,E1 -11552.126,E2 -11552.126} C_VEL
LIN {X 0,Y 390.08,Z 575.896,A -85,B 0,C 180,E1 -11555.208,E2 -11555.208} C_VEL
LIN {X 0,Y 390.09,Z 575.896,A -85,B 0,C 180,E1 -11559.093,E2 -11559.093} C_VEL
LIN {X 0,Y 390.118,Z 575.885,A -85,B 0,C 180,E1 -11562.388,E2 -11562.388} C_VEL
LIN {X 0,Y 390.115,Z 575.959,A -85,B 0,C 180,E1 -11564.636,E2 -11564.636} C_VEL
LIN {X 0,Y 391.81,Z 584.176,A -85,B 0,C 180,E1 -11567.921,E2 -11567.921} C_VEL
LIN {X 0,Y 393.368,Z 591.799,A -85,B 0,C 180,E1 -11570.788,E2 -11570.788} C_VEL
LIN {X 0,Y 394.14,Z 597.187,A -85,B 0,C 180,E1 -11572.682,E2 -11572.682} C_VEL
LIN {X 0,Y 393.703,Z 602.939,A -85,B 0,C 180,E1 -11574.54,E2 -11574.54} C_VEL
LIN {X 0,Y 392.513,Z 614.492,A -85,B 0,C 180,E1 -11578.117,E2 -11578.117} C_VEL
LIN {X 0,Y 391.58,Z 626.011,A -85,B 0,C 180,E1 -11581.576,E2 -11581.576} C_VEL
LIN {X 0,Y 390.787,Z 637.759,A -85,B 0,C 180,E1 -11585.001,E2 -11585.001} C_VEL
LIN {X 0,Y 390.162,Z 649.406,A -85,B 0,C 180,E1 -11588.331,E2 -11588.331} C_VEL
LIN {X 0,Y 389.825,Z 658.693,A -85,B 0,C 180,E1 -11590.911,E2 -11590.911} C_VEL
LIN {X 0,Y 392.402,Z 676.438,A -85,B 0,C 180,E1 -11591.596,E2 -11591.596} C_VEL
LIN {X 0,Y 393.257,Z 689.555,A -85,B 0,C 180,E1 -11592.22,E2 -11592.22} C_VEL
LIN {X 0,Y 393.919,Z 702.333,A -85,B 0,C 180,E1 -11593.014,E2 -11593.014} C_VEL
LIN {X 0,Y 393.162,Z 714.385,A -85,B 0,C 180,E1 -11593.916,E2 -11593.916} C_VEL
LIN {X 0,Y 392.19,Z 725.395,A -85,B 0,C 180,E1 -11594.941,E2 -11594.941} C_VEL
LIN {X 0,Y 391.421,Z 734.689,A -85,B 0,C 180,E1 -11596.003,E2 -11596.003} C_VEL
LIN {X 0,Y 390.63,Z 743.848,A -85,B 0,C 180,E1 -11597.269,E2 -11597.269} C_VEL
LIN {X 0,Y 389.894,Z 752.996,A -85,B 0,C 180,E1 -11598.828,E2 -11598.828} C_VEL
LIN {X 0,Y 389.425,Z 760.456,A -85,B 0,C 180,E1 -11600.391,E2 -11600.391} C_VEL
LIN {X 0,Y 389.163,Z 765.509,A -85,B 0,C 180,E1 -11601.694,E2 -11601.694} C_VEL
LIN {X 0,Y 388.942,Z 770.425,A -85,B 0,C 180,E1 -11603.256,E2 -11603.256} C_VEL
LIN {X 0,Y 388.918,Z 774.183,A -85,B 0,C 180,E1 -11604.817,E2 -11604.817} C_VEL
LIN {X 0,Y 388.846,Z 776.096,A -85,B 0,C 180,E1 -11605.855,E2 -11605.855} C_VEL
LIN {X 0,Y 388.868,Z 777.549,A -85,B 0,C 180,E1 -11606.893,E2 -11606.893} C_VEL
LIN {X 0,Y 388.935,Z 778.593,A -85,B 0,C 180,E1 -11607.93,E2 -11607.93} C_VEL
LIN {X 0,Y 388.924,Z 779.215,A -85,B 0,C 180,E1 -11608.966,E2 -11608.966} C_VEL
LIN {X 0,Y 388.95,Z 779.373,A -85,B 0,C 180,E1 -11610.001,E2 -11610.001} C_VEL
LIN {X 0,Y 388.935,Z 779.118,A -85,B 0,C 180,E1 -11611.036,E2 -11611.036} C_VEL
LIN {X 0,Y 388.937,Z 778.456,A -85,B 0,C 180,E1 -11612.072,E2 -11612.072} C_VEL
LIN {X 0,Y 388.883,Z 777.335,A -85,B 0,C 180,E1 -11613.109,E2 -11613.109} C_VEL
LIN {X 0,Y 388.896,Z 774.829,A -85,B 0,C 180,E1 -11614.665,E2 -11614.665} C_VEL
LIN {X 0,Y 388.914,Z 770.96,A -85,B 0,C 180,E1 -11616.331,E2 -11616.331} C_VEL
LIN {X 0,Y 389.06,Z 766.51,A -85,B 0,C 180,E1 -11617.787,E2 -11617.787} C_VEL
LIN {X 0,Y 389.348,Z 760.467,A -85,B 0,C 180,E1 -11619.35,E2 -11619.35} C_VEL
LIN {X 0,Y 389.748,Z 752.913,A -85,B 0,C 180,E1 -11620.915,E2 -11620.915} C_VEL
LIN {X 0,Y 390.327,Z 745.19,A -85,B 0,C 180,E1 -11622.215,E2 -11622.215} C_VEL
LIN {X 0,Y 391.061,Z 735.757,A -85,B 0,C 180,E1 -11623.512,E2 -11623.512} C_VEL
LIN {X 0,Y 391.605,Z 726.592,A -85,B 0,C 180,E1 -11624.553,E2 -11624.553} C_VEL
LIN {X 0,Y 392.402,Z 715.358,A -85,B 0,C 180,E1 -11625.585,E2 -11625.585} C_VEL
LIN {X 0,Y 393.255,Z 702.695,A -85,B 0,C 180,E1 -11626.482,E2 -11626.482} C_VEL
LIN {X 0,Y 392.434,Z 691.33,A -85,B 0,C 180,E1 -11627.14,E2 -11627.14} C_VEL
LIN {X 0,Y 391.378,Z 677.93,A -85,B 0,C 180,E1 -11627.706,E2 -11627.706} C_VEL
LIN {X 0,Y 389.671,Z 660.124,A -85,B 0,C 180,E1 -11628.297,E2 -11628.297} C_VEL
LIN {X 0,Y 390.059,Z 647.922,A -85,B 0,C 180,E1 -11631.677,E2 -11631.677} C_VEL
LIN {X 0,Y 390.63,Z 635.997,A -85,B 0,C 180,E1 -11635.012,E2 -11635.012} C_VEL
LIN {X 0,Y 391.4,Z 623.203,A -85,B 0,C 180,E1 -11638.627,E2 -11638.627} C_VEL
LIN {X 0,Y 392.151,Z 611.862,A -85,B 0,C 180,E1 -11641.918,E2 -11641.918} C_VEL
LIN {X 0,Y 393.029,Z 600.686,A -85,B 0,C 180,E1 -11645.218,E2 -11645.218} C_VEL
LIN {X 0,Y 393.442,Z 595.181,A -85,B 0,C 180,E1 -11646.886,E2 -11646.886} C_VEL
LIN {X 0,Y 392.91,Z 590.488,A -85,B 0,C 180,E1 -11648.39,E2 -11648.39} C_VEL
LIN {X 0,Y 390.842,Z 579.589,A -85,B 0,C 180,E1 -11652.076,E2 -11652.076} C_VEL
LIN {X 0,Y 390.073,Z 575.898,A -85,B 0,C 180,E1 -11653.43,E2 -11653.43} C_VEL
LIN {X 0,Y 390.062,Z 575.9,A -85,B 0,C 180,E1 -11656.79,E2 -11656.79} C_VEL
LIN {X 0,Y 390.062,Z 575.899,A -85,B 0,C 180,E1 -11659.561,E2 -11659.561} C_VEL
LIN {X 0,Y 390.051,Z 575.901,A -85,B 0,C 180,E1 -11662.449,E2 -11662.449} C_VEL
LIN {X 0,Y 390.073,Z 575.897,A -85,B 0,C 180,E1 -11666.045,E2 -11666.045} C_VEL
LIN {X 0,Y 390.051,Z 575.899,A -85,B 0,C 180,E1 -11669.869,E2 -11669.869} C_VEL
LIN {X 0,Y 390.118,Z 575.888,A -85,B 0,C 180,E1 -11673.232,E2 -11673.232} C_VEL
LIN {X 0,Y 390.111,Z 575.891,A -85,B 0,C 180,E1 -11676.75,E2 -11676.75} C_VEL
LIN {X 0,Y 390.109,Z 575.892,A -85,B 0,C 180,E1 -11679.983,E2 -11679.983} C_VEL
LIN {X 0,Y 390.143,Z 575.885,A -85,B 0,C 180,E1 -11683.248,E2 -11683.248} C_VEL
LIN {X 0,Y 390.199,Z 575.882,A -85,B 0,C 180,E1 -11686.561,E2 -11686.561} C_VEL
LIN {X 0,Y 390.209,Z 575.88,A -85,B 0,C 180,E1 -11690.671,E2 -11690.671} C_VEL
LIN {X 0,Y 390.323,Z 575.865,A -85,B 0,C 180,E1 -11692.759,E2 -11692.759} C_VEL
LIN {X 0,Y 390.23,Z 575.876,A -85,B 0,C 180,E1 -11694.833,E2 -11694.833} C_VEL
LIN {X 0,Y 390.421,Z 575.853,A -85,B 0,C 180,E1 -11697.936,E2 -11697.936} C_VEL
LIN {X 0,Y 390.554,Z 575.836,A -85,B 0,C 180,E1 -11700,E2 -11700} C_VEL
LIN {X 0,Y 390.313,Z 575.865,A -85,B 0,C 180,E1 -11703.096,E2 -11703.096} C_VEL
LIN {X 0,Y 390.313,Z 575.864,A -85,B 0,C 180,E1 -11706.638,E2 -11706.638} C_VEL
LIN {X 0,Y 390.208,Z 575.877,A -85,B 0,C 180,E1 -11709.328,E2 -11709.328} C_VEL
LIN {X 0,Y 390.198,Z 575.878,A -85,B 0,C 180,E1 -11713.438,E2 -11713.438} C_VEL
LIN {X 0,Y 390.152,Z 575.884,A -85,B 0,C 180,E1 -11717.307,E2 -11717.307} C_VEL
LIN {X 0,Y 390.09,Z 575.896,A -85,B 0,C 180,E1 -11720.469,E2 -11720.469} C_VEL
LIN {X 0,Y 390.092,Z 575.891,A -85,B 0,C 180,E1 -11723.35,E2 -11723.35} C_VEL
LIN {X 0,Y 390.116,Z 575.891,A -85,B 0,C 180,E1 -11726.768,E2 -11726.768} C_VEL
LIN {X 0,Y 390.041,Z 575.902,A -85,B 0,C 180,E1 -11730.299,E2 -11730.299} C_VEL
LIN {X 0,Y 390.07,Z 575.896,A -85,B 0,C 180,E1 -11734.024,E2 -11734.024} C_VEL
LIN {X 0,Y 390.047,Z 575.897,A -85,B 0,C 180,E1 -11737.551,E2 -11737.551} C_VEL
LIN {X 0,Y 390.058,Z 575.898,A -85,B 0,C 180,E1 -11740.821,E2 -11740.821} C_VEL
LIN {X 0,Y 390.059,Z 575.897,A -85,B 0,C 180,E1 -11743.886,E2 -11743.886} C_VEL
LIN {X 0,Y 390.061,Z 575.898,A -85,B 0,C 180,E1 -11746.789,E2 -11746.789} C_VEL
LIN {X 0,Y 390.058,Z 575.895,A -85,B 0,C 180,E1 -11749.56,E2 -11749.56} C_VEL
LIN {X 0,Y 390.044,Z 575.902,A -85,B 0,C 180,E1 -11752.448,E2 -11752.448} C_VEL
LIN {X 0,Y 390.068,Z 575.896,A -85,B 0,C 180,E1 -11756.044,E2 -11756.044} C_VEL
LIN {X 0,Y 390.047,Z 575.898,A -85,B 0,C 180,E1 -11759.868,E2 -11759.868} C_VEL
LIN {X 0,Y 390.114,Z 575.889,A -85,B 0,C 180,E1 -11763.231,E2 -11763.231} C_VEL
LIN {X 0,Y 390.107,Z 575.893,A -85,B 0,C 180,E1 -11766.749,E2 -11766.749} C_VEL
LIN {X 0,Y 390.104,Z 575.891,A -85,B 0,C 180,E1 -11769.982,E2 -11769.982} C_VEL
LIN {X 0,Y 390.138,Z 575.886,A -85,B 0,C 180,E1 -11773.247,E2 -11773.247} C_VEL
